// ---- GVLs/GVL10_VAR_PRG.TcGVL
(* Variables for program blocks *)
VAR_GLOBAL PERSISTENT
	
	nPowerFailureCounter					:UINT;
	
END_VAR
VAR_GLOBAL
	
	(* PLC start detected *)
	bFirstCycleDetected						:BOOL;
	bMachineSequenzAktiv					:BOOL;		(* PLC startup done (LED test) program in cyclic mode *)

	(* Clock generator *)
	bClock500ms								:BOOL;		(* Clock 500ms on/off *)
	bClock1s								:BOOL;		(* Clock 1s on/off *)
	bClock2s								:BOOL;		(* Clock 2s on/off *)
	bRisingEdge500ms						:BOOL;		(* Rising edge all 500ms over one cycle *)
	bRisingEdge1s							:BOOL;		(* Edge after 1s over a cycle *)
	bRisingEdge2s							:BOOL;		(* Edge after 2s over a cycle *)

END_VAR
(* End *)

// ---- GVLs/GVL20_Axis.TcGVL
(* GVL20_Axis - Global variables axis *)
{attribute 'TcContextName' := 'PlcTask'}
VAR_GLOBAL
	
(* Axis 1 inputs and outputs *)
	stAxis1									:AXIS_REF;

(* Axis 2 inputs and outputs *)
	stAxis2									:AXIS_REF;

(* Axis 3 - 4 (AX5203) inputs and outputs *)
	nAxis3TorqueFeedback			AT%I*	:INT;		(* Axis 3 current +/- 1000 *)
	nAxis4TorqueFeedback			AT%I*	:INT;		(* Axis 4 current +/- 1000 *)

	nAX5203DigitalInputs			AT%I*	:UINT;		(* Digital inputs AX5000
															BIT 0 - servo reference cam (axis 3)
															BIT 1 - servo reference cam (axis 4)
															BIT 2 - switch S26
															BIT 3 - switch S27 *)

	nAX5203DigitalOutputs			AT%Q*	:UINT;		(* Digital output AX5000 
															BIT 7 - Led H27 *)
	
	stAxis3									:AXIS_REF;
	stAxis4									:AXIS_REF;

(* Axis 5 (Handwheel) inputs and outputs *)
	stAxis5									:AXIS_REF;

END_VAR
(* End *)

// ---- GVLs/GVL30_DiagnosticEtherCAT.TcGVL
(* GVL30_DiagnosticEtherCAT *)
{attribute 'TcContextName' := 'PlcTask'}
VAR_GLOBAL

	fbDiagnosticEtherCAT					:FB_DiagnosticEtherCAT;

END_VAR
(* End *)

// ---- POUs/Sample OOP Conveyor/Device And Station Blocks/GVL_Products.TcGVL
VAR_GLOBAL
	arrParts : ARRAY[0..100] OF ST_PartData; // all the products currently in the machine
END_VAR

// ---- POUs/Sample UML SC/GVL_UML.TcGVL
VAR_GLOBAL
	nCounterInit				: INT;
	nCounterSaveInitSettings	: INT;
	nCounterClearXml			: INT;
	nCounterFillXml				: INT;
	nCounterSaveXml				: INT;
	nCounterClearText			: INT;
	nCounterFillText			: INT;
	nCounterSaveText			: INT;
	nCounterGetMasterID			: INT;
	nCounterGetClientID			: INT;
	nCounterSendToMaster		: INT;
	nCounterSendToClient		: INT;
	
	bMasterFirst				: BOOL;
	bClientFirst				: BOOL;
END_VAR

// ---- POUs/Sample OOP/Cylinder/ICylinder.TcIO
INTERFACE ICylinder

METHOD M_StateMachine : BOOL
VAR_INPUT
	bPosLeftReq  : BOOL;
	bPosRightReq : BOOL;
END_VAR
VAR_OUTPUT
	bAtLeftPos   : BOOL;
	bAtRightPos  : BOOL; 
END_VAR
END_METHOD

PROPERTY P_TimerValue : LREAL
GET
END_GET
SET
END_SET
END_PROPERTY

END_INTERFACE

// ---- POUs/Sample OOP/Regulator/IRegulator.TcIO
INTERFACE IRegulator

METHOD M_Active : UINT
VAR_INPUT
	(* controller input  *)
	fSetpointValue			: LREAL;		// setpoint value
	fActualValue			: LREAL;		// actual value
	bReset					: BOOL;			// reset flag
	(* controller values *)
	stRegParams				: ST_RegParams;
END_VAR
VAR_OUTPUT
	fCtrlOutput				: LREAL;		// controller output command
END_VAR
END_METHOD

PROPERTY P_Error : BOOL
GET
END_GET
SET
END_SET
END_PROPERTY

END_INTERFACE

// ---- POUs/Sample OOP/Table/Axis/IAxis.TcIO
INTERFACE IAxis

METHOD M_Diag : BOOL
VAR_INPUT
END_VAR
VAR_OUTPUT
	bNcError 	: BOOL;
	bDrvError 	: BOOL;
	iNcErrorId	: UDINT;
END_VAR
END_METHOD

METHOD M_Enable : BOOL
VAR_INPUT
	bEnable 	: BOOL;
	fOverride	: LREAL;
END_VAR
END_METHOD

METHOD M_HardwareDiag : BOOL
VAR_INPUT
	bExecute : BOOL;
END_VAR
END_METHOD

METHOD M_HardwareReset : BOOL
VAR_INPUT
	bExecute : BOOL;
END_VAR
END_METHOD

{attribute 'InstanceVar'}
METHOD M_Move : BOOL
VAR_INPUT
	bExecute	: BOOL;
	eMoveCmd	: E_MoveCmd;
	fVelocity	: LREAL;
	fPosition	: LREAL;
END_VAR
END_METHOD

METHOD M_Reset : BOOL
VAR_INPUT
	bExecute 	: BOOL;
END_VAR
END_METHOD

END_INTERFACE

// ---- POUs/Sample OOP Conveyor/Axis Blocks/I_Axis.TcIO
INTERFACE I_Axis

METHOD M_Disable : UDINT
VAR_INPUT
	bDisable : BOOL;
END_VAR
//The result of the method is an unsigned double integer
// 0 = idle 
// 1 = busy
// 3 = complete
// Any other number = Error
END_METHOD

METHOD M_Enable : UDINT
VAR_INPUT
	bEnable :BOOL;
END_VAR
//The result of the method is an unsigned double integer
// 0 = idle 
// 1 = busy
// 3 = complete
// Any other number = Error
END_METHOD

METHOD M_HardwareReset : UDINT
VAR_INPUT
	bReset:BOOL;
END_VAR
//The result of the method is an unsigned double integer
// 0 = idle 
// 1 = busy
// 3 = complete
// Any other number = Error number
END_METHOD

METHOD M_Jog : UDINT
VAR_INPUT
	bJogFwd : BOOL;
	bJogBwd : BOOL;
	fJogSpeed : LREAL;
END_VAR
//The result of the method is an unsigned double integer
// 0 = idle 
// 1 = busy
// 3 = complete
// Any other number = Error
END_METHOD

METHOD M_Reset : UDINT
VAR_INPUT
	bReset : BOOL;
END_VAR
//The result of the method is an unsigned double integer
// 0 = idle 
// 1 = busy
// 3 = complete
// Any other number = Error
END_METHOD

METHOD M_Speed : UDINT
VAR_INPUT
	bMoveVelocity : BOOL;
	fSpeed : LREAL;
END_VAR
//The result of the method is an unsigned double integer
// 0 = idle 
// 1 = busy
// 3 = complete
// Any other number = Error
END_METHOD

METHOD M_Stop : UDINT
VAR_INPUT
	bStop : BOOL;
END_VAR
//The result of the method is an unsigned double integer
// 0 = idle 
// 1 = busy
// 3 = complete
// Any other number = Error
END_METHOD

PROPERTY P_CurrentPosition : LREAL
GET
END_GET
SET
END_SET
END_PROPERTY

PROPERTY P_CurrentSpeed : LREAL
GET
END_GET
SET
END_SET
END_PROPERTY

PROPERTY P_Error : BOOL
GET
END_GET
SET
END_SET
END_PROPERTY

PROPERTY P_ErrorID : UDINT
GET
END_GET
SET
END_SET
END_PROPERTY

PROPERTY P_Ready : BOOL
GET
END_GET
SET
END_SET
END_PROPERTY

END_INTERFACE

// ---- POUs/Sample OOP Conveyor/Device And Station Blocks/I_Mode.TcIO
INTERFACE I_Mode

METHOD M_Auto : UDINT
VAR_INPUT
	bRequestAutoMode : BOOL;
END_VAR
END_METHOD

METHOD M_Disable : UDINT
VAR_INPUT
	bDisable : BOOL;
END_VAR
END_METHOD

METHOD M_Manual : UDINT
VAR_INPUT
	bRequestManualMode: BOOL;
END_VAR
END_METHOD

METHOD M_Reset : UDINT
VAR_INPUT
	bRequestReset:BOOL;
END_VAR
END_METHOD

PROPERTY P_CurrentState : E_Modes
GET
END_GET
SET
END_SET
END_PROPERTY

END_INTERFACE

// ---- POUs/RT Monitor/extMarksPrg.TcPOU
PROGRAM extMarksPrg
VAR
    fbLogMark	: FB_RTMon_LogMarkBase;	
	
	// user defined context
	idModule1 : UINT := 10001;	

		
	// Marks
	markCounter  : ST_RTMon_MarkDef := (nContextId := idModule1, nGroupId := 1, nEventId := 0); 
END_VAR

//fbLogMark.LogMarkEx(markCounter, TcMarkOption.Start OR TcMarkOption.RefToCaller);
IF GVL.fbCrititcalSection.Enter() THEN
	GVL.iGlobalCounter:=GVL.iGlobalCounter+1;
	ConsumeTime(50);
    GVL.fbCrititcalSection.Leave();
END_IF
//fbLogMark.LogMarkEx(markCounter, TcMarkOption.Stop OR TcMarkOption.RefToCaller);

END_PROGRAM

// ---- POUs/RT Monitor/logging/ConsumeTime.TcPOU
FUNCTION ConsumeTime : bool
VAR_INPUT
	DelayUs 	: UDINT;
END_VAR
VAR
	fbGetTime	: GETCPUACCOUNT;
	tStart		: UDINT;
	tNow		: UDINT;
END_VAR

fbGetTime(cpuAccountDW => tStart);
tNow := tStart;

WHILE (tNow - tStart) < DelayUs*10 DO
	fbGetTime(cpuAccountDW => tNow);
END_WHILE

END_FUNCTION

// ---- POUs/MainPOUs/MAIN.TcPOU
PROGRAM MAIN
(*******************************************************************************************************
Title				:	Main program 
Description			:	Calling the created subroutines (Task 1ms)
Version / Date		:	1.0.0 / 23.05.2016 / created program (Version progress see below)

Supported hardware	: 	Demo-Rack (LAGE version)

Used Documentation	:	
Documentation	
Version/Date 		:	

Required libraries 	: 	Please look in the "References" folder
********************************************************************************************************)
VAR
	
(* Cycle counter *)
	nCycleCounter							:UDINT;

(* act_SUps - 1s UPS - Uninterruptible power supply *)
	fbSUps									:FB_S_UPS_CX51x0 := (eUpsMode:=eSUPS_WrPersistData_Shutdown);
	bPowerFailDetect						:BOOL;

(* act_SystemStart *)
	eStateSystemStartSeq					:E_SystemStartupSequence;
	eSystemStartSeqErrStep					:E_SystemStartupSequence := eSystemStart_NoError;
	bSystemStartErr							:BOOL;
	bSystemStartEnd							:BOOL;
	fbTimerSystemStart						:TON;


(*******************************************************************************************************
Version / Date / Description:
1.0.0   / 23.05.2016 / created program
********************************************************************************************************)
(* End *)

	{attribute 'TcContextName':='PlcTask'}
	iCounter AT %Q*		: DINT;
	
	//fbMC2				: FB_MC2;
	//fbNCI				: FB_NCI;
	fbOOPAxisTable		: FB_OOPAxisTable;
	fbOOPCylReg			: FB_OOPCylinderRegulator;
	fbOOPConveyor		: FB_OOPConveyor;
	
	{attribute 'TcAnalytics'}
	fbScope				: FB_GenerateData;
	fbUmlSc				: FB_UML_SC_Composite;
	fbUmlSc_Lamp		: FB_UML_SC_Lamp;

	fbModeChangeTimer	: TON := (PT := T#60S);
	nRemainingModeTime	: UDINT;
	
	eSampleMode			: E_SampleMode;	
	eSampleModeMC2		: E_SampleMode;	
	eSampleModeNCI		: E_SampleMode;	
	eSampleModeOOP		: E_SampleMode;	
	eSampleModeOOPConv	: E_SampleMode;	

	nRadioButton		: INT;
	AxisRef				: ARRAY [1..iMAX_AXES_REF] OF AXIS_REF;			// axis reference (process data plc/nc)
	
	{attribute 'TcContextName':='PlcTask'}
	wFrmXWcState_MAIN AT %I*	: WORD; 			// link to NC-task related ethercat frame state (Frm0WcState)
	x1: WORD;
	
	fblog : FB_RTMon_LogMark;

END_VAR

(* MAIN - 1ms *)

(* THIS CODE IS ONLY AN EXAMPLE - YOU HAVE TO CHECK APTITUDE FOR YOUR APPLICATION *)

(* Cycle counter *)
	nCycleCounter := nCycleCounter + 1;


(* 1s USV *)
	act_SUps();


(* Startup detect *)
	IF TwinCAT_SystemInfoVarList._TaskInfo[GETCURTASKINDEXEX()].FirstCycle
	THEN
		bFirstCycleDetected	:= TRUE;
	END_IF


(* Startup- or machine sequence *)
	IF bFirstCycleDetected
	THEN
	(* Startup sequenz *)
		act_SystemStart();

		IF bSystemStartEnd
		THEN
			bFirstCycleDetected := FALSE;
			bMachineSequenzAktiv := TRUE;
		END_IF

	ELSIF bMachineSequenzAktiv
	THEN
	(* Machine sequenz *)
		(* Test general *)
			GeneralPlc();
		
		(* Test blinker *)
			Blinker();

		(* Test clock generator *)
			ClockGenerator();
		
		(* Test axis *)
			AxisGeneral();
			Axis1();
			Axis2();
			Axis3();
			Axis4();
			stAxis5.ReadStatus();

		(* Test EtherCAT diacnostic *)
			DiagnosticEtherCAT();
			
		(* Test - XFC - extrem fast control *)	
			DcTimes();
			AnalogOutputOversampling();
			PositionCamTimeStampAxis2();
			SignalLengthMeasurementCamAxis2();
			TouchProbeTimeStampCamAxis2();

		(* Test TwinSAFE *)	
			TwinSAFE();
		
	END_IF

(* End *)

iCounter := iCounter + 1;

//switch mode (MC2, NCI, OOP)
A_ModeSwitch();

(*//call MC2 sample
fblog.LogStart(1,0); //added this
fbMC2(AxisRef := AxisRef, eSampleModeIn := eSampleMode, eSampleModeOut => eSampleModeMC2);
fblog.LogStop(1,0); // added this*)


//call NCI sample
fblog.LogStart(2,0); //added this
NCI();
//fbNCI(AxisRef := AxisRef, eSampleModeIn := eSampleMode, eSampleModeOut => eSampleModeNCI);
fblog.LogStop(2,0);

//Call Cam Table Sample
CamTable();

//Call External Setpoint Generator Sample
Ext_SP_Gen();

//call OOP sample
fblog.LogStart(3,0);
fbOOPAxisTable(AxisRef := AxisRef, eSampleModeIn := eSampleMode, eSampleModeOut => eSampleModeOOP);
fbOOPCylReg();
fblog.LogStop(3,0);

//call OOP conveyor sample
fblog.logstart(4,0);
fbOOPConveyor(AxisRef := AxisRef, eSampleModeIn := eSampleMode, eSampleModeOut => eSampleModeOOPConv);
fblog.logstop(4,0);

//call language samples
fblog.LogMark(5,0);
MAIN_CFC();					//continuous flow chart
fblog.LogMark(5,1);
MAIN_CFC_PageOriented();	//continuous flow chart, page oriented
fblog.LogMark(5,2);
MAIN_FBD_IL_LD();			//use language switching via menu "FBD/IL/LD, function block diagram, instruction list, ladder logic 
fblog.LogMark(5,3);
MAIN_SFC();					//sequential flow chart 
fblog.LogMark(5,4);
MAIN_ST();					//structured text
fblog.LogStop(5,0);


//call UML SC composite sample
fblog.LogStart(6,0);
fbUmlSc();
fbUmlSc_Lamp();
fblog.LogStop(6,0);

x1 := wFrmXWcState_MAIN;

//Call TwinSAFE Program
TwinSAFE();

//Call IoT Program
IoT_JSON_XML();

//Call Database Server Sample
CSVSample();

ACTION A_ModeSwitch:
//decide for an active motion sample
fbModeChangeTimer(IN := TRUE);
nRemainingModeTime := TIME_TO_UDINT(fbModeChangeTimer.PT-fbModeChangeTimer.ET)/1000;

IF fbModeChangeTimer.Q OR (eSampleMode = eSMode_Idle) OR (nRadioButton > 0) THEN
	//switch if ready 
	
	IF (eSampleModeMC2 = eSMode_Idle) AND (eSampleModeNCI = eSMode_Idle) AND (eSampleModeOOP = eSMode_Idle) AND (eSampleModeOOPConv = eSMode_Idle) THEN
		//ready to switch
		fbModeChangeTimer(IN := FALSE);
		
		CASE eSampleMode OF
		eSMode_Idle:
			CASE nRadioButton OF
			1:
				eSampleMode := eSMode_MC2_Req;
			2:			
				eSampleMode := eSMode_NCI_Req;
			3:			
				eSampleMode := eSMode_OOP_Req;
			4:			
				eSampleMode := eSMode_OOPConv_Req;
			ELSE //idle
				eSampleMode := eSMode_MC2_Req;
			END_CASE
			
		eSMode_MC2_Req:
			CASE nRadioButton OF
			1:
				eSampleMode := eSMode_MC2_Req;
			2:			
				eSampleMode := eSMode_NCI_Req;
			3:			
				eSampleMode := eSMode_OOP_Req;
			4:			
				eSampleMode := eSMode_OOPConv_Req;
			ELSE //idle
				eSampleMode := eSMode_NCI_Req;
			END_CASE
			
		eSMode_NCI_Req:
			CASE nRadioButton OF
			1:
				eSampleMode := eSMode_MC2_Req;
			2:			
				eSampleMode := eSMode_NCI_Req;
			3:			
				eSampleMode := eSMode_OOP_Req;
			4:			
				eSampleMode := eSMode_OOPConv_Req;
			ELSE //idle
				eSampleMode := eSMode_OOP_Req;
			END_CASE
			
		eSMode_OOP_Req:
			CASE nRadioButton OF
			1:
				eSampleMode := eSMode_MC2_Req;
			2:			
				eSampleMode := eSMode_NCI_Req;
			3:			
				eSampleMode := eSMode_OOP_Req;
			4:			
				eSampleMode := eSMode_OOPConv_Req;
			ELSE //idle
				eSampleMode := eSMode_MC2_Req;
			END_CASE
			
		eSMode_OOPConv_Req:
			CASE nRadioButton OF
			1:
				eSampleMode := eSMode_MC2_Req;
			2:			
				eSampleMode := eSMode_NCI_Req;
			3:			
				eSampleMode := eSMode_OOP_Req;
			4:			
				eSampleMode := eSMode_OOPConv_Req;
			ELSE //idle
				eSampleMode := eSMode_MC2_Req;
			END_CASE
			
		ELSE
			eSampleMode := eSMode_MC2_Req;
		END_CASE
		
		nRadioButton := 0;
	END_IF 
END_IF
END_ACTION

ACTION act_SUps:
(* Aktion - 1s UPS - Uninterruptible power supply *)

	fbSUps(); (* see instance declaration for initalisation of eUpsMode parameter *) 

	(*
	Default Values of FB_S_UPS_CX51x0-Inputs:
						sNetID 			:=	'' -> local netid
						iPLCPort 		:=	AMSPORT_R0_PLC_RTS1 -> 801 = 1st PLC Runtime 
						iUPSPort		:=	16#588 -> Port for reading Power State of UPS
						tTimeout 		:=	DEFAULT_ADS_TIMEOUT -> 5S
						eUpsMode 		:=	eSUPS_WrPersistData_Shutdown -> writing persistent data + shutdown
						ePersistentMode :=	SPDM_2PASS -> All data is from same plc cycle, cycletime exceeds possible. Plc stops with the shutdown, a few cycles after writing persistent data. 
						tRecoverTime 	:=	T#10s -> 10s power to recover from short power failure before eSUPS_PowerOK is reported (in mode eSUPS_WrPersistData_NoShutdown/eSUPS_CheckPowerStatus)

	eUpsMode =							in case of powerfailure:
	 	eSUPS_WrPersistData_Shutdown 	->	writing of persistent data + shutdown
	 	eSUPS_WrPersistData_NoShutdown 	->	writing of PERSISTENT data, no shutdown
	 	eSUPS_CheckPowerStatus 			->	reports powerfailure without ACTION (no writing, no shutdown) 
	 	eSUPS_ImmediateShutdown 		->	skips writing of data, immediate shutdown
	*)	

(* Power fail detected *)
	IF fbSUps.bPowerFailDetect
		AND NOT bPowerFailDetect
	THEN
	
		(* Count the power failures *)
		nPowerFailureCounter := nPowerFailureCounter + 1;
		bPowerFailDetect	 := TRUE;
	
	ELSE

		IF NOT fbSUps.bPowerFailDetect
		THEN
			bPowerFailDetect:=FALSE;
		END_IF

	END_IF

(* End *)
END_ACTION

ACTION act_SystemStart:
(* Aktion system start *)

	CASE eStateSystemStartSeq OF

	
		eSystemStart_Start			: 	(* Waiting for start *)
		
				eStateSystemStartSeq := eSystemStart_Init;

				
		eSystemStart_Init			:	(* Initialize *)

				fbTimerSystemStart(IN := FALSE);
				eStateSystemStartSeq := eSystemStart_LedOn;

				
		eSystemStart_LedOn			:	(* Sequence Leds on *)

				fbTimerSystemStart(	
					IN := TRUE,
					PT := T#2250MS);

				bLedH10	:=	fbTimerSystemStart.ET > T#250MS;
				bLedH20 :=  bLedH10;
				bLedH31 :=  bLedH10;
				bLedH11	:=	fbTimerSystemStart.ET > T#500MS;
				bLedH21 :=  bLedH11;
				bLedH32 :=  bLedH11;
				bLedH12	:=	fbTimerSystemStart.ET > T#750MS;
				bLedH22 :=  bLedH12;
				bLedH33 :=  bLedH12;
				bLedH13	:=	fbTimerSystemStart.ET > T#1000MS;
				bLedH23 :=  bLedH13;
				bLedH14	:=	fbTimerSystemStart.ET > T#1250MS;
				bLedH24 :=  bLedH14;
				bLedH15	:=	fbTimerSystemStart.ET > T#1500MS;
				bLedH25 :=  bLedH15;
				bLedH16	:=	fbTimerSystemStart.ET > T#1750MS;
				bLedH26 :=  bLedH16;
				bLedH17	:=	fbTimerSystemStart.ET > T#2000MS;
				nAX5203DigitalOutputs.7 :=  bLedH17;

				IF fbTimerSystemStart.Q
				THEN
					fbTimerSystemStart(IN := FALSE);
					eStateSystemStartSeq := eSystemStart_LedOff;
				ELSIF FALSE
				THEN
					(* If error then notice the step *)
					eSystemStartSeqErrStep := eStateSystemStartSeq;
					eStateSystemStartSeq   := eSystemStart_ErrorStep;
				END_IF

				
		eSystemStart_LedOff			:	(* Sequence Leds off *)

				fbTimerSystemStart(	
					IN := TRUE,
					PT := T#2250MS);

				bLedH10	:=	fbTimerSystemStart.ET < T#250MS;
				bLedH20 :=  bLedH10;
				bLedH31 :=  bLedH10;
				bLedH11	:=	fbTimerSystemStart.ET < T#500MS;
				bLedH21 :=  bLedH11;
				bLedH32 :=  bLedH11;
				bLedH12	:=	fbTimerSystemStart.ET < T#750MS;
				bLedH22 :=  bLedH12;
				bLedH33 :=  bLedH12;
				bLedH13	:=	fbTimerSystemStart.ET < T#1000MS;
				bLedH23 :=  bLedH13;
				bLedH14	:=	fbTimerSystemStart.ET < T#1250MS;
				bLedH24 :=  bLedH14;
				bLedH15	:=	fbTimerSystemStart.ET < T#1500MS;
				bLedH25 :=  bLedH15;
				bLedH16	:=	fbTimerSystemStart.ET < T#1750MS;
				bLedH26 :=  bLedH16;
				bLedH17	:=	fbTimerSystemStart.ET < T#2000MS;
				nAX5203DigitalOutputs.7 :=  bLedH17;
									
				IF fbTimerSystemStart.Q
				THEN
					eStateSystemStartSeq := eSystemStart_Done;
				ELSIF FALSE
				THEN
					(* If error then notice the step *)
					eSystemStartSeqErrStep := eStateSystemStartSeq;
					eStateSystemStartSeq   := eSystemStart_ErrorStep;
				END_IF

				
		eSystemStart_Done			:	(* System start done *)

				bSystemStartEnd := TRUE;

				
		eSystemStart_ErrorStep		:	(* Error on system start *)

				bSystemStartErr := TRUE;

				IF FALSE
				THEN
					bSystemStartErr        := FALSE;
					eSystemStartSeqErrStep := eSystemStart_NoError;
					eStateSystemStartSeq   := eSystemStart_Start;
				END_IF 

	ELSE
		
		(* If not a valid step is active, then put on start *)
		eSystemStartSeqErrStep := eSystemStart_NoError;
		eStateSystemStartSeq   := eSystemStart_Start;
	
	END_CASE

(* End *)
END_ACTION

END_PROGRAM

// ---- POUs/Sample OOP/FB_OOPAxisTable.TcPOU
FUNCTION_BLOCK FB_OOPAxisTable
VAR_INPUT
	eSampleModeIn	: E_SampleMode;	
END_VAR
VAR_IN_OUT
	AxisRef			: ARRAY [1..iMAX_AXES_REF] OF AXIS_REF;			// axis reference (process data plc/nc)
END_VAR
VAR_OUTPUT
	eSampleModeOut	: E_SampleMode;	
END_VAR
VAR
	iCounter 			: DINT;
END_VAR	
VAR
	//instances of axes FBs (of type FB_NcAxes or derived from FB_NcAxis, like AX5000, Servo Termins, Stepper, DC, ...)
	fbAX5000Axis1	: FB_AX5000Axis;
	fbAX5000Axis2	: FB_AX5000Axis;
	fbNcAxis		: FB_NcAxis;
		
	//interface pointers
	ipAxisX			: IAxis;
	ipAxisY			: IAxis;
	ipAxisZ			: IAxis;

	//device
	fbTable			: FB_Table;
	bExecute		: BOOL;
	bBusy			: BOOL;
	
	Timer			: TON := (PT := T#3s);
END_VAR

iCounter := iCounter + 1;

IF (eSampleModeIn = eSMode_OOP_Req) OR (eSampleModeOut = eSMode_OOP_Act) THEN
	//assign axes instances to the interface pointers
	ipAxisX := fbAX5000Axis1;
	ipAxisY := fbAX5000Axis2;
	ipAxisZ	:= fbNcAxis;
	
	//call axes with their axes references
	fbAX5000Axis1(sAxis	:= AxisRef[1]);
	fbAX5000Axis2(sAxis	:= AxisRef[2]);
	fbNcAxis(sAxis	:= AxisRef[3]);
	
	Timer(IN := TRUE);
	IF Timer.Q THEN
		Timer(IN := FALSE);
		bExecute := TRUE;
	END_IF
	
	//call device that uses axes via interface, therefore the axis type does not matter anymore
	fbTable(
		fbServoAxisX := ipAxisX,
		fbServoAxisY := ipAxisY,
		fbServoAxisZ := ipAxisZ,
		bExecute	 := bExecute,
		bBusy		 => bBusy
	);
		
	bExecute := FALSE;

	IF bBusy THEN
		eSampleModeOut := eSMode_OOP_Act;
	ELSE
		eSampleModeOut := eSMode_Idle;
	END_IF
END_IF

END_FUNCTION_BLOCK

// ---- POUs/Sample OOP/Table/Axis/FB_AX5000Axis.TcPOU
FUNCTION_BLOCK FB_AX5000Axis EXTENDS FB_NcAxis
VAR_INPUT
END_VAR
VAR_OUTPUT
END_VAR
VAR
	fbSoEReadDiagNumber : FB_SoEReadDiagNumber;
	iDiagNumber			: UDINT;
	fbSoEReset			: FB_SoEReset;
END_VAR

METHOD M_HardwareDiag : BOOL
VAR_INPUT
	bExecute	: BOOL;
END_VAR
//get hardware diag
CASE eCurState OF
eAxisState_Idle:
	IF bExecute AND NOT bExecHWDiag_  THEN
		fbSoEReadDiagNumber(
			NetId:= '', 
			Execute:= TRUE, 
			Axis:= sAxis, 
		);
		eCurState := eAxisState_Diag;
	END_IF

eAxisState_Diag:
	fbSoEReadDiagNumber(
		NetId:= '', 
		Execute:= TRUE, 
		Axis:= sAxis, 
	);
	IF NOT fbSoEReadDiagNumber.Busy  THEN
		fbSoEReadDiagNumber(
			Execute:= FALSE, 
			Axis:= sAxis, 
			DiagNumber=> iDiagNumber
		);
		eCurState := eAxisState_Idle;
	END_IF
	
END_CASE

M_HardwareDiag 	:= eCurState <> eAxisState_Idle;	
bExecHWDiag_	:= bExecute;
END_METHOD

METHOD M_HardwareReset : BOOL
VAR_INPUT
	bExecute	: BOOL;
END_VAR
//reset axis
CASE eCurState OF
eAxisState_Idle:
	IF bExecute AND NOT bExecHWRes_ THEN
		fbSoEReset(
			NetId:= '', 
			Execute:= TRUE, 
			Axis:= sAxis, 
		);
		eCurState := eAxisState_Reset;
	END_IF

eAxisState_Reset:
	fbSoEReset(
		NetId:= '', 
		Execute:= TRUE, 
		Axis:= sAxis, 
	);
	IF NOT fbSoEReset.Busy THEN
		fbSoEReset(
			Execute:= FALSE, 
			Axis:= sAxis, 
		);
		eCurState := eAxisState_Idle;
	END_IF

END_CASE

M_HardwareReset := eCurState <> eAxisState_Idle;	
bExecHWRes_		:= bExecute;
END_METHOD

END_FUNCTION_BLOCK

// ---- POUs/Sample OOP/Table/Axis/FB_NcAxis.TcPOU
FUNCTION_BLOCK FB_NcAxis IMPLEMENTS IAxis
VAR_IN_OUT
	sAxis		: AXIS_REF;
END_VAR
VAR_INPUT
END_VAR
VAR_OUTPUT
	bActive		: BOOL;
	bBusy		: BOOL;
	bDone		: BOOL;
	bError		: BOOL;
	iErrorId	: UDINT;
	eCurState	: E_AxisState;
END_VAR
VAR
	//PLCopen FBs for axes
	fbMcPower	: MC_Power;
	fbMcReset	: MC_Reset;
	fbMcMoveAbs	: MC_MoveAbsolute;
	fbMcMoveMod	: MC_MoveModulo;
	fbMcMoveRel	: MC_MoveRelative;
	fbMcMoveVel	: MC_MoveVelocity;

	//rising edge detection
	bExecMove_	: BOOL;
	bExecHWDiag_: BOOL;
	bExecHWRes_	: BOOL;
	bExecReset_	: BOOL;
END_VAR

;

METHOD M_Diag : BOOL
VAR_INPUT
END_VAR
VAR_OUTPUT
	bNcError 	: BOOL;
	bDrvError 	: BOOL;
	iNcErrorId	: UDINT;
END_VAR
//get axis diag
sAxis.ReadStatus();
bNcError	:= sAxis.NcToPlc.StateDWord.31;
bDrvError	:= sAxis.NcToPlc.StateDWord.28;
iNcErrorId	:= sAxis.NcToPlc.ErrorCode;
M_Diag 		:= bNcError OR bDrvError OR (iNcErrorId <> 0);
END_METHOD

METHOD M_Enable : BOOL
VAR_INPUT
	bEnable		: BOOL;
	fOverride	: LREAL;
END_VAR
//enable axis
fbMcPower(
	Enable		:= bEnable, 	Enable_Positive	:= bEnable,	Enable_Negative	:= bEnable, 
	Override	:= fOverride, 	Axis			:= sAxis
);
M_Enable := fbMcPower.Status;
END_METHOD

METHOD M_HardwareDiag : BOOL
VAR_INPUT
	bExecute	: BOOL;
END_VAR
//get hardware diag --> overwrite method if necessary
CASE eCurState OF
eAxisState_Idle:
	IF bExecute AND NOT bExecHWDiag_ THEN
		eCurState := eAxisState_Diag;
	END_IF

eAxisState_Diag:
		eCurState := eAxisState_Idle;

END_CASE

M_HardwareDiag 	:= eCurState <> eAxisState_Idle;	
bExecHWDiag_	:= bExecute;
END_METHOD

METHOD M_HardwareReset : BOOL
VAR_INPUT
	bExecute	: BOOL;
END_VAR
//hardware reset axis --> overwrite method if necessary
CASE eCurState OF
eAxisState_Idle:
	IF bExecute AND NOT bExecHWRes_ THEN
		eCurState := eAxisState_Reset;
	END_IF

eAxisState_Reset:
		eCurState := eAxisState_Idle;

END_CASE

M_HardwareReset := eCurState <> eAxisState_Idle;	
bExecHWRes_		:= bExecute;
END_METHOD

METHOD M_Move : BOOL
VAR_INPUT
	bExecute	: BOOL;
	eMoveCmd	: E_MoveCmd;
	fVelocity	: LREAL;
	fPosition	: LREAL;
END_VAR
//move axis
CASE eCurState OF
eAxisState_Idle:	
	IF bExecute AND NOT bExecMove_ THEN
		CASE eMoveCmd OF
		eCmd_MoveAbsolute:
			fbMcMoveAbs(
				Execute	:= bExecute, 	Position:= fPosition,	Velocity:= fVelocity, 
				Axis	:= sAxis, 		Done	=> bDone,		Busy	=> bBusy, 
				Active	=> bActive, 	Error	=> bError,		ErrorID	=> iErrorId
			);
			eCurState := eAxisState_Move;
		
		eCmd_MoveModulo:
			fbMcMoveMod(
				Execute	:= bExecute, 	Position:= fPosition,	Velocity:= fVelocity, 
				Axis	:= sAxis, 		Done	=> bDone, 		Busy	=> bBusy, 
				Active	=> bActive, 	Error	=> bError,		ErrorID	=> iErrorId
			);
			eCurState := eAxisState_Move;
		
		eCmd_MoveRelative:
			fbMcMoveRel(
				Execute	:= bExecute, 	Distance:= fPosition,	Velocity:= fVelocity, 
				Axis	:= sAxis, 		Done	=> bDone,		Busy	=> bBusy, 
				Active	=> bActive, 	Error	=> bError,		ErrorID	=> iErrorId
			);
			eCurState := eAxisState_Move;
		
		eCmd_MoveVelocity:
			fbMcMoveVel(
				Execute	:= bExecute, 	Velocity:= fVelocity,	Axis	:= sAxis, 
				InVelocity=> bDone,		Busy	=> bBusy,		Active	=> bActive, 
				Error	=> bError, 		ErrorID	=> iErrorId,	Busy	=> bBusy,
				Active	=> bActive,		Error	=> bError,		ErrorID	=> iErrorId
			);		
			eCurState := eAxisState_Move;
		END_CASE
	END_IF
		
eAxisState_Move:
	CASE eMoveCmd OF
	eCmd_MoveAbsolute:
		fbMcMoveAbs(
			Execute	:= TRUE, 		Position:= fPosition,	Velocity:= fVelocity, 
			Axis	:= sAxis, 		Done	=> bDone,		Busy	=> bBusy, 
			Active	=> bActive, 	Error	=> bError, 		ErrorID	=> iErrorId
		);
		IF bDone OR bError THEN
			fbMcMoveAbs(Execute	:= FALSE,Axis := sAxis); 
			eCurState := eAxisState_Idle;
		END_IF
	
	eCmd_MoveModulo:
		fbMcMoveMod(
			Execute	:= TRUE, 		Position:= fPosition,	Velocity:= fVelocity, 
			Axis	:= sAxis, 		Done	=> bDone,		Busy	=> bBusy, 
			Active	=> bActive, 	Error	=> bError,		ErrorID	=> iErrorId
		);
		IF bDone OR bError THEN
			fbMcMoveMod(Execute	:= FALSE,Axis := sAxis); 
			eCurState := eAxisState_Idle;
		END_IF
	
	eCmd_MoveRelative:
		fbMcMoveRel(
			Execute	:= TRUE, 		Distance:= fPosition,	Velocity:= fVelocity, 
			Axis	:= sAxis, 		Done	=> bDone,		Busy	=> bBusy, 
			Active	=> bActive, 	Error	=> bError,		ErrorID	=> iErrorId
		);
		IF bDone OR bError THEN
			fbMcMoveRel(Execute	:= FALSE,Axis := sAxis); 
			eCurState := eAxisState_Idle;
		END_IF
	
	eCmd_MoveVelocity:
		fbMcMoveVel(
			Execute	:= TRUE, 		Velocity:= fVelocity,	Axis	:= sAxis, 
			InVelocity=> bDone,		Busy	=> bBusy,		Active	=> bActive, 
			Error	=> bError, 		ErrorID	=> iErrorId,	Busy	=> bBusy, 		
			Active	=> bActive,		Error	=> bError,		ErrorID	=> iErrorId
		);		
		IF bDone OR bError THEN
			fbMcMoveVel(Execute	:= FALSE,Axis := sAxis); 
			eCurState := eAxisState_Idle;
		END_IF
	END_CASE
END_CASE

M_Move 		:= (eCurState <> eAxisState_Idle);
bExecMove_	:= bExecute;
END_METHOD

METHOD M_Reset : BOOL
VAR_INPUT
	bExecute	: BOOL;
END_VAR
//reset nc axis
CASE eCurState OF
eAxisState_Idle:
	IF bExecute AND NOT bExecReset_ THEN
		fbMcReset(
			Execute	:= bExecute, 	Axis	:= sAxis,	Done	=> bDone, 
			Busy	=> bBusy, 		Error	=> bError,	ErrorID	=> iErrorId 
		);
		eCurState := eAxisState_Reset;
	END_IF

eAxisState_Reset:
	fbMcReset(
		Execute	:= FALSE, 	Axis	:= sAxis,	Done	=> bDone, 
		Busy	=> bBusy, 	Error	=> bError,	ErrorID	=> iErrorId 
	);
	IF fbMcReset.Done OR fbMcReset.Error THEN
		eCurState := eAxisState_Idle;
	END_IF
END_CASE

M_Reset 	:= eCurState <> eAxisState_Idle;	
bExecReset_	:= bExecute;
END_METHOD

END_FUNCTION_BLOCK

// ---- POUs/Sample OOP/Table/FB_Table.TcPOU
FUNCTION_BLOCK FB_Table
VAR_IN_OUT
	fbServoAxisX	: IAxis; //Pass the reference to ANY block that uses FB_NcAxis as a base class
	fbServoAxisY	: IAxis; //Pass the reference to ANY block that uses FB_NcAxis as a base class
	fbServoAxisZ	: IAxis; //Pass the reference to ANY block that uses FB_NcAxis as a base class
END_VAR
VAR_INPUT
	bEnable			: BOOL	:= TRUE;
	fOverride		: LREAL	:= 100;
	bExecute		: BOOL;
END_VAR
VAR_OUTPUT
	bEnabled		: BOOL;
	bBusy			: BOOL;
	bError			: BOOL;
END_VAR
VAR
	iState			: INT;
	bExecute_		: BOOL;

	eCurStateAxisX	: E_AxisState;
	bEnabledAxisX	: BOOL;
	bBusyAxisX		: BOOL;
	bErrorAxisX		: BOOL;

	eCurStateAxisY	: E_AxisState;
	bEnabledAxisY	: BOOL;
	bBusyAxisY		: BOOL;
	bErrorAxisY		: BOOL;

	eCurStateAxisZ	: E_AxisState;
	bEnabledAxisZ	: BOOL;
	bBusyAxisZ		: BOOL;
	bErrorAxisZ		: BOOL;
END_VAR

//NC axes can be used independent of axes type (AX5000, stepper, analog axis, ...) incl. hardware reset and diagnostic  

//enable axes
bEnabledAxisX 	:= fbServoAxisX.M_Enable(bEnable:= bEnable, fOverride:= fOverride);
bEnabledAxisY 	:= fbServoAxisY.M_Enable(bEnable:= bEnable, fOverride:= fOverride);
bEnabledAxisZ 	:= fbServoAxisZ.M_Enable(bEnable:= bEnable, fOverride:= fOverride);
bEnabled		:= bEnabledAxisX AND bEnabledAxisY AND bEnabledAxisZ;

//check for cyclic diagnostics
bErrorAxisX		:= fbServoAxisX.M_Diag();
bErrorAxisY		:= fbServoAxisY.M_Diag();
bErrorAxisZ		:= fbServoAxisZ.M_Diag();
bError			:= bError OR bErrorAxisX OR bErrorAxisY OR bErrorAxisZ;

//state machine
CASE iState OF
	0:	//idle state
		IF (bExecute AND NOT bExecute_) THEN
			IF bError THEN
				iState := 10;
			ELSIF bEnabled THEN
				iState := iState + 1;
			END_IF
		END_IF	
		
	1:	//move x 200, y 200, z 200
		bBusyAxisX := fbServoAxisX.M_Move(bExecute:= TRUE, eMoveCmd:= eCmd_MoveAbsolute, fVelocity:= 100.0, fPosition:= 200.0);
		bBusyAxisY := fbServoAxisY.M_Move(bExecute:= TRUE, eMoveCmd:= eCmd_MoveAbsolute, fVelocity:= 100.0, fPosition:= 200.0);
		bBusyAxisZ := fbServoAxisZ.M_Move(bExecute:= TRUE, eMoveCmd:= eCmd_MoveAbsolute, fVelocity:= 100.0, fPosition:= 200.0);
		IF NOT bBusyAxisX AND NOT bBusyAxisY AND NOT bBusyAxisZ THEN
			bBusyAxisX := fbServoAxisX.M_Move(bExecute:= FALSE, eMoveCmd:= eCmd_MoveAbsolute, fVelocity:= 100.0, fPosition:= 200.0);
			bBusyAxisY := fbServoAxisY.M_Move(bExecute:= FALSE, eMoveCmd:= eCmd_MoveAbsolute, fVelocity:= 100.0, fPosition:= 200.0);
			bBusyAxisZ := fbServoAxisZ.M_Move(bExecute:= FALSE, eMoveCmd:= eCmd_MoveAbsolute, fVelocity:= 100.0, fPosition:= 200.0);
			iState := iState + 1;
		END_IF
		
	2:	//move x 100, y 300
		bBusyAxisX := fbServoAxisX.M_Move(bExecute:= TRUE, eMoveCmd:= eCmd_MoveAbsolute, fVelocity:= 150.0, fPosition:= 100.0);
		bBusyAxisY := fbServoAxisY.M_Move(bExecute:= TRUE, eMoveCmd:= eCmd_MoveAbsolute, fVelocity:= 150.0, fPosition:= 300.0);
		IF NOT bBusyAxisX AND NOT bBusyAxisY THEN
			bBusyAxisX := fbServoAxisX.M_Move(bExecute:= FALSE, eMoveCmd:= eCmd_MoveAbsolute, fVelocity:= 150.0, fPosition:= 100.0);
			bBusyAxisY := fbServoAxisY.M_Move(bExecute:= FALSE, eMoveCmd:= eCmd_MoveAbsolute, fVelocity:= 150.0, fPosition:= 300.0);
			iState := iState + 1;
		END_IF
		
	3:	//move x 0, y 0, z 0
		bBusyAxisX := fbServoAxisX.M_Move(bExecute:= TRUE, eMoveCmd:= eCmd_MoveAbsolute, fVelocity:= 50.0, fPosition:= 0.0);
		bBusyAxisY := fbServoAxisY.M_Move(bExecute:= TRUE, eMoveCmd:= eCmd_MoveAbsolute, fVelocity:= 150.0, fPosition:= 0.0);
		bBusyAxisZ := fbServoAxisZ.M_Move(bExecute:= TRUE, eMoveCmd:= eCmd_MoveAbsolute, fVelocity:= 150.0, fPosition:= 0.0);
		IF NOT bBusyAxisX AND NOT bBusyAxisY AND NOT bBusyAxisZ THEN
			bBusyAxisX := fbServoAxisX.M_Move(bExecute:= FALSE, eMoveCmd:= eCmd_MoveAbsolute, fVelocity:= 50.0, fPosition:= 0.0);
			bBusyAxisY := fbServoAxisY.M_Move(bExecute:= FALSE, eMoveCmd:= eCmd_MoveAbsolute, fVelocity:= 150.0, fPosition:= 0.0);
			bBusyAxisZ := fbServoAxisZ.M_Move(bExecute:= FALSE, eMoveCmd:= eCmd_MoveAbsolute, fVelocity:= 150.0, fPosition:= 0.0);
			iState := 0;
		END_IF
		
	10:	//hardware diag
		bBusyAxisX := fbServoAxisX.M_HardwareDiag(bExecute:= TRUE);
		bBusyAxisY := fbServoAxisY.M_HardwareDiag(bExecute:= TRUE);
		bBusyAxisZ := fbServoAxisZ.M_HardwareDiag(bExecute:= TRUE);
		IF NOT bBusyAxisX AND NOT bBusyAxisY AND NOT bBusyAxisZ THEN
			bBusyAxisX := fbServoAxisX.M_HardwareDiag(bExecute:= FALSE);
			bBusyAxisY := fbServoAxisY.M_HardwareDiag(bExecute:= FALSE);
			bBusyAxisZ := fbServoAxisZ.M_HardwareDiag(bExecute:= FALSE);
			iState := iState + 1;
		END_IF

	11:	//hardware reset
		bBusyAxisX := fbServoAxisX.M_HardwareReset(bExecute:= TRUE);
		bBusyAxisY := fbServoAxisY.M_HardwareReset(bExecute:= TRUE);
		bBusyAxisZ := fbServoAxisZ.M_HardwareReset(bExecute:= TRUE);
		IF NOT bBusyAxisX AND NOT bBusyAxisY AND NOT bBusyAxisZ THEN
			bBusyAxisX := fbServoAxisX.M_HardwareReset(bExecute:= FALSE);
			bBusyAxisY := fbServoAxisY.M_HardwareReset(bExecute:= FALSE);
			bBusyAxisZ := fbServoAxisZ.M_HardwareReset(bExecute:= FALSE);
			iState := iState + 1;
		END_IF
		
	12:	//nc reset
		bBusyAxisX := fbServoAxisX.M_Reset(bExecute:= TRUE);
		bBusyAxisY := fbServoAxisY.M_Reset(bExecute:= TRUE);
		bBusyAxisZ := fbServoAxisZ.M_Reset(bExecute:= TRUE);
		IF NOT bBusyAxisX AND NOT bBusyAxisY AND NOT bBusyAxisZ THEN
			bBusyAxisX := fbServoAxisX.M_Reset(bExecute:= FALSE);
			bBusyAxisY := fbServoAxisY.M_Reset(bExecute:= FALSE);
			bBusyAxisZ := fbServoAxisZ.M_Reset(bExecute:= FALSE);
			bError := FALSE;
			iState := 0;
		END_IF

END_CASE

bBusy		:= bBusyAxisX OR bBusyAxisY OR bBusyAxisZ;
bExecute_ 	:= bExecute;

END_FUNCTION_BLOCK

// ---- POUs/Sample OOP/FB_OOPCylinderRegulator.TcPOU
FUNCTION_BLOCK FB_OOPCylinderRegulator
VAR
	iCounter 				: DINT;	

	(* Interface Instance of ICylinder *)
	ipCylinder 				: ICylinder;

	(* cylinder with feedback and without/with diag  *)
	fbCylinder 				: FB_Cylinder;		//instance of cylinder without diag 
	fbCylinderDiag			: FB_CylinderDiag;	//instance of cylinder with diag
	bEnableDiag				: BOOL := FALSE;	//enable diagnose cylinder
	bDiagAvailable			: BOOL;				//diag is enabled
	lrTimerValue 			: LREAL := 0.2;		//simulation time [s]
	tTimeOutDiag 			: TIME := T#1S100MS;//diagnose timeout
	bDiag	 				: BOOL;				//diagnose feedback

	(* cmds/state *)
	bMoveToLeftReq AT %I*	: BOOL;		//cmd move to left side
	bMoveToRightReq AT %I*	: BOOL;		//cmd move to right side
	bCylinderAtLeft AT %Q* 	: BOOL;		//state at left side
	bCylinderAtRight AT %Q*	: BOOL;		//state at left side


	(* Interface Instance of IRegulator *)
	ipRegulator 		: IRegulator;

	(* P/PID Regulator *)
	fbBasicP			: FB_BasicP;		// instance of P-Controller
	fbBasicPID			: FB_BasicPID;		// instance of PID-Controller
	bEnablePID			: BOOL;				// enable PID
	bPIDEnabled			: BOOL;				// PID enabled
	fSetpointValue		: LREAL;			// setpoint value
	fActualValue		: LREAL;			// actual value
	bReset				: BOOL;				// reset flag
	stRegParams			: ST_RegParams;		// parameters for the regulator
	fCtrlOutput			: LREAL;			// controller output command
	bErrorFlag			: BOOL;				// controller error
	

	(* common *)
	Timer 				: TON := (PT := T#5S);	 //simulation timer
	bInit 				: BOOL := TRUE;
	bSimulation			: BOOL := TRUE;
	bMoveToLeftReqSim 	: BOOL := TRUE;		//cmd move to left side
	bMoveToRightReqSim	: BOOL := FALSE;	//cmd move to right side
	nErrorStatus		: UINT;				//controller error output (0: no error; >0:error)
	fNoise				: LREAL;
	bNoiseUp			: BOOL;
END_VAR

iCounter := iCounter + 1;

(* initialization *)
IF bInit THEN
	A_Init();
END_IF
A_Simulation();


(* --- CYLINDER --- assign FB instance to the interface instance *)
IF NOT bEnableDiag THEN
	ipCylinder := fbCylinder;
	bDiagAvailable := FALSE;
ELSE
	ipCylinder := fbCylinderDiag;
	bDiagAvailable := FALSE;
END_IF

(* access property via interface instance *)
ipCylinder.P_TimerValue := lrTimerValue; //Set property
lrTimerValue := ipCylinder.P_TimerValue; //Get property

(* call FB via interface instance *)
bDiag := ipCylinder.M_StateMachine(
	bPosLeftReq 	:= bMoveToLeftReq,	
	bPosRightReq 	:= bMoveToRightReq,
	bAtLeftPos		=> bCylinderAtLeft,
	bAtRightPos		=> bCylinderAtRight,
);


(* --- REGULATOR --- assign FB instance to the interface instance *)
IF bEnablePID THEN
	ipRegulator := fbBasicPID;
	bPIDEnabled := TRUE;
ELSE
	ipRegulator := fbBasicP;
	bPIDEnabled := FALSE;
END_IF

(* call FB via interface instance *)
nErrorStatus := ipRegulator.M_Active(
	fSetpointValue	:= fSetpointValue,
	fActualValue	:= fActualValue,
	bReset			:= bReset,
	stRegParams		:= stRegParams,
	fCtrlOutput		=> fCtrlOutput
);

(* access property via interface instance *)
bErrorFlag := ipRegulator.P_Error; 	//Get
ipRegulator.P_Error := FALSE; 		//Set

ACTION A_Init:
bInit := FALSE;

fbCylinderDiag(tTimeOut := tTimeOutDiag);

stRegParams.fCtrlCycleTime := 0.010; 
stRegParams.fKp := 1.9; 
stRegParams.fTd := 0; 
stRegParams.fTn := 0; 
stRegParams.fTv := 0; 
fSetpointValue	:= 100;
fNoise 			:= 2.2;
bNoiseUp 		:= TRUE;
END_ACTION

ACTION A_Simulation:
Timer(IN := TRUE);

IF Timer.Q THEN
	Timer(IN := FALSE);
	IF bMoveToLeftReqSim THEN
		bMoveToLeftReqSim 	:= FALSE;
		bMoveToRightReqSim 	:= TRUE;	//cmd move to right side
 	ELSE
		bMoveToLeftReqSim 	:= TRUE;	//cmd move to left side
		bMoveToRightReqSim	:= FALSE;
	END_IF
END_IF

IF bSimulation THEN
	MEMCPY(ADR(bMoveToLeftReq), ADR(bMoveToLeftReqSim), SIZEOF(bMoveToLeftReq));
	MEMCPY(ADR(bMoveToRightReq), ADR(bMoveToRightReqSim), SIZEOF(bMoveToRightReq));

	IF fNoise >= 10 THEN
		bNoiseUp := FALSE;
	ELSIF fNoise <= -10 THEN
		bNoiseUp := TRUE;
	END_IF

	IF bNoiseUp THEN
		fNoise := fNoise + 0.01;
	ELSE
		fNoise := fNoise - 0.01;
	END_IF
	fNoise := LIMIT(-11.0, fNoise, 11.0);
  
	fActualValue := fActualValue + LIMIT(-100,fCtrlOutput,100) + fNoise;
END_IF
END_ACTION

END_FUNCTION_BLOCK

// ---- POUs/Sample OOP/Cylinder/FB_Cylinder.TcPOU
FUNCTION_BLOCK FB_Cylinder IMPLEMENTS ICylinder //regular FB that additionally implements an interface "ICylinder"
VAR_INPUT
END_VAR
VAR_OUTPUT
END_VAR
VAR
	//internal TIME variable that is being accessed via property "P_Timervalue" (Get/Set)
	tTimerValue 	: TIME := T#500MS;

	iState			: INT;
	bAtLeftPosFbk	: BOOL;
	bAtRightPosFbk	: BOOL;
	TimerReach 		: TON;
	TimerStart 		: TON;
END_VAR

;

METHOD M_StateMachine : BOOL
VAR_INPUT
	bPosLeftReq	: BOOL;
	bPosRightReq: BOOL;
END_VAR
VAR_OUTPUT
	bAtLeftPos	: BOOL;
	bAtRightPos	: BOOL;
END_VAR
// variables of a method are temporary and therefore cleared in teh next cycle 
// variables of the FB can be used for keeping variable values over many PLC cycles
(* simple cylinder with feedback  *)
CASE iState OF
0: (* at left pos *)
	bAtLeftPosFbk := TRUE;
	bAtRightPosFbk := FALSE;
	
	IF bPosRightReq THEN
		TimerStart(IN := FALSE);
		TimerReach(IN := FALSE);
		iState := iState + 1;
	END_IF

1: (* start motion to right side *)
	 TimerStart(IN := TRUE, PT := tTimerValue);
	 IF TimerStart.Q THEN
		bAtLeftPosFbk := FALSE;
		TimerStart(IN := FALSE);
		TimerReach(IN := TRUE);
		iState := iState + 1;
	 END_IF

2: (* moving *)
	 TimerReach(IN := TRUE, PT := tTimerValue);
	 IF TimerReach.Q THEN
		bAtRightPosFbk := TRUE;
		TimerReach(IN := FALSE);
		iState := iState + 1;
	 END_IF

3: (* right pos reached *)
	bAtLeftPosFbk := FALSE;
	bAtRightPosFbk := TRUE;
	
	IF bPosLeftReq THEN
		TimerStart(IN := FALSE);
		TimerReach(IN := FALSE);
		iState := iState + 1;
	END_IF

4: (* start motion to left side *)
	 TimerStart(IN := TRUE, PT := tTimerValue);
	 IF TimerStart.Q THEN
		bAtRightPosFbk := FALSE;
		TimerStart(IN := FALSE);
		TimerReach(IN := TRUE);
		iState := iState + 1;
	 END_IF

5: (* moving *)
	 TimerReach(IN := TRUE, PT := tTimerValue);
	 IF TimerReach.Q THEN
		bAtLeftPosFbk := TRUE;
		TimerReach(IN := FALSE);
		iState := 0;
	 END_IF
END_CASE

bAtLeftPos 		:= bAtLeftPosFbk;
bAtRightPos 	:= bAtRightPosFbk;

M_StateMachine 	:= FALSE;
END_METHOD

PROPERTY P_TimerValue : LREAL //encapsulates internal variable tTimerValue
GET
//read property (returns value of of internal variable)
P_TimerValue := TIME_TO_LREAL(tTimerValue) * LREAL#0.001; //convert ms (TIME) to s (LREAL)
END_GET
SET
//write property (set value of of internal variable)
tTimerValue := LREAL_TO_TIME(P_TimerValue * LREAL#1000); //convert s (LREAL) to ms (TIME)
END_SET
END_PROPERTY

END_FUNCTION_BLOCK

// ---- POUs/Sample OOP/Cylinder/FB_CylinderDiag.TcPOU
FUNCTION_BLOCK FB_CylinderDiag EXTENDS FB_Cylinder
VAR_INPUT
	tTimeOut 	  : TIME;
END_VAR
VAR
	WatchDogTimer : TON;
END_VAR

;

METHOD M_Diag : BOOL
VAR_INPUT
END_VAR
IF (iState = 0) OR (iState = 3) THEN
	WatchDogTimer(IN := FALSE, PT := tTimeOut);
ELSE
	WatchDogTimer(IN := TRUE, PT := tTimeOut);
END_IF

M_Diag := WatchDogTimer.Q;
END_METHOD

METHOD M_StateMachine : BOOL
VAR_INPUT
	bPosLeftReq  : BOOL;
	bPosRightReq : BOOL;
END_VAR
VAR_OUTPUT
	bAtLeftPos  : BOOL;
	bAtRightPos : BOOL; 
END_VAR
//call M_StateMachine of base class (FB_Cylinder) via 'SUPER^.' (access to things of FB_CylinderDiag via 'THIS^.')  
SUPER^.M_StateMachine(
	bPosLeftReq 	:= bPosLeftReq,	
	bPosRightReq 	:= bPosRightReq,
	bAtLeftPos		=> bAtLeftPos,
	bAtRightPos		=> bAtRightPos,
);

//additional diagnosis
M_StateMachine 		:= M_Diag();
END_METHOD

END_FUNCTION_BLOCK

// ---- POUs/Sample OOP/Regulator/FB_BasicP.TcPOU
FUNCTION_BLOCK FB_BasicP IMPLEMENTS IRegulator //regular FB that additionally implements an interface "IRegulator" as P-Controller
VAR CONSTANT
	nERR_NOERROR			: UINT := 0;	// no error
	nERR_INVALIDPARAM		: UINT := 1;	// invalid parameter
	nERR_INVALIDCYCLETIME	: UINT := 2;	// invalid cycle time				
END_VAR
VAR
	(* STATIC VARIABLE *)
	(* Internal Variable *)
	fE						: LREAL := 0.0;	// error input
	fE_1					: LREAL := 0.0;	// error input z^(-1)
	fY						: LREAL := 0.0;	// control output
	fY_1					: LREAL := 0.0;	// control output  z^(-1)
	fYP						: LREAL := 0.0;	// P-part
	nErrorStatus			: UINT;			// controller error output (0: no error; >0:error)
	(* Internal Parameter *)
	bInit					: BOOL	:= TRUE;// initialization flag for first cycle
	fCtrlCycleTimeOld		: LREAL	:= 0.0;
	fKpOld					: LREAL	:= 0.0;
END_VAR

;

METHOD M_Active 	: UINT
VAR_INPUT
	(* controller input  *)
	fSetpointValue	: LREAL;		// setpoint value
	fActualValue	: LREAL;		// actual value
	bReset			: BOOL;			// reset flag
	(* controller values *)
	stRegParams		: ST_RegParams;
END_VAR
VAR_OUTPUT
	fCtrlOutput		: LREAL;		// controller output command
END_VAR
(* init necessary? *)
IF (stRegParams.fCtrlCycleTime <> fCtrlCycleTimeOld) OR (stRegParams.fKp <> fKpOld) THEN
	bInit := TRUE;
END_IF

(* controller init *)
IF bInit OR bReset THEN
	(* reset internal and external variables *)
	fE	:= fE_1		:= 0.0;
	fY	:= fY_1		:= 0.0;
	fYP	:= 0.0;
	fCtrlOutput		:= 0.0;
	nErrorStatus	:= nERR_NOERROR;

	(* check cycle time parameter: (CycleTime > 0 AND CycleTme <= 60) *)
	IF ( stRegParams.fCtrlCycleTime <= 0) THEN
		nErrorStatus := nERR_INVALIDCYCLETIME;
		M_Active := nErrorStatus;
		RETURN;
	END_IF;

	(* reset *)
	IF bReset THEN
		M_Active := nErrorStatus;
		RETURN;
	END_IF

	(* set internal init flag *)
	fCtrlCycleTimeOld 	:= stRegParams.fCtrlCycleTime;
	fKpOld 				:= stRegParams.fKp;
	bInit				:= FALSE;
END_IF;

(* 3. save old variable *)
fE_1		:= fE;
fY_1		:= fY;

(* 4. set error/deviation input *)
fE	:= fSetpointValue - fActualValue;

(* 5. YP-part *)
fYp		:= stRegParams.fKp * fE;

(* 8. Ysum = YP *)
fY	:= fYP;

(* 10. set controller output *)
fCtrlOutput := fY;

M_Active := nErrorStatus;
END_METHOD

PROPERTY P_Error : BOOL
GET
P_Error := (nErrorStatus <> 0); // get error status
END_GET
SET
nErrorStatus := 0; // clear error status
END_SET
END_PROPERTY

END_FUNCTION_BLOCK

// ---- POUs/Sample OOP/Regulator/FB_BasicPID.TcPOU
FUNCTION_BLOCK FB_BasicPID IMPLEMENTS IRegulator //regular FB that additionally implements an interface "IRegulator" as PID-Controller
VAR CONSTANT
	nERR_NOERROR			: UINT := 0;	// no error
	nERR_INVALIDPARAM		: UINT := 1;	// invalid parameter
	nERR_INVALIDCYCLETIME	: UINT := 2;	// invalid cycle time				
END_VAR
VAR
	(*
		                       1               Tv * s						
	  	G(s) = Kp * ( 1 + ------------ + --------------- )				
	                         Tn * s       1 + Td * s					
	*)

	(* STATIC VARIABLE *)
	(* Internal Variable *)
	fE						: LREAL := 0.0;	// error input
	fE_1					: LREAL := 0.0;	// error input z^(-1)
	fY						: LREAL := 0.0;	// control output
	fY_1					: LREAL := 0.0;	// control output  z^(-1)
	fYP						: LREAL := 0.0;	// P-part
	fYI						: LREAL := 0.0;	// I-part			
	fYI_1					: LREAL := 0.0;	// I-part  z^(-1)	
	fYD						: LREAL := 0.0;	// D-T1-part		
	fYD_1					: LREAL := 0.0;	// D-T1-part  z^(-1)
	nErrorStatus			: UINT;			// controller error output (0: no error; >0:error)
	(* Internal Parameter *)
	bInit					: BOOL	:= TRUE;// initialization flag for first cycle
	bIsIPart				: BOOL	:= FALSE;// I-part active ?
	bIsDPart				: BOOL	:= FALSE;// D-part active ?
	fDi						: LREAL	:= 0.0;	// internal I param
	fDd						: LREAL	:= 0.0;	// internal D param
	fCd						: LREAL	:= 0.0;	// internal D param
	fCtrlCycleTimeOld		: LREAL	:= 0.0;
	fKpOld					: LREAL	:= 0.0;
	fTnOld					: LREAL	:= 0.0;
	fTvOld					: LREAL	:= 0.0;
	fTdOld					: LREAL	:= 0.0;
END_VAR

;

METHOD M_Active 	: UINT
VAR_INPUT
	(* controller input  *)
	fSetpointValue	: LREAL;		// setpoint value
	fActualValue	: LREAL;		// actual value
	bReset			: BOOL;			// reset flag
	(* controller values *)
	stRegParams		: ST_RegParams;
END_VAR
VAR_OUTPUT
	fCtrlOutput		: LREAL;		// controller output command
END_VAR
(* init necessary? *)
IF (stRegParams.fCtrlCycleTime <> fCtrlCycleTimeOld) OR (stRegParams.fKp <> fKpOld) OR (stRegParams.fTn <> fTnOld) 
	OR (stRegParams.fTv <> fTvOld) OR (stRegParams.fTd <> fTdOld) THEN
	
	bInit := TRUE;
END_IF

(* controller init *)
IF bInit OR bReset THEN
	(* reset internal and external variables *)
	fE	:= fE_1		:= 0.0;
	fY	:= fY_1		:= 0.0;
	fYP	:= 0.0;
	fYI	:= fYI_1	:= 0.0;
	fYD	:= fYD_1	:= 0.0;
	fCtrlOutput		:= 0.0;
	bIsIPart		:= FALSE;
	bIsDPart		:= FALSE;
	fCtrlOutput		:= 0.0;
	nErrorStatus	:= nERR_NOERROR;

	(* check cycle time parameter: (CycleTime > 0 AND CycleTme <= 60) *)
	IF ( stRegParams.fCtrlCycleTime <= 0) 	THEN
		nErrorStatus := nERR_INVALIDCYCLETIME;
		M_Active := nErrorStatus;
		RETURN;
	END_IF;

	(* check controller parameters: (Tn, Tv, Td >= 0) *)
	IF ( (stRegParams.fTn < 0) OR (stRegParams.fTv < 0) OR (stRegParams.fTd < 0) ) THEN
		nErrorStatus := nERR_INVALIDPARAM;
		M_Active := nErrorStatus;
		RETURN;
	END_IF;

	(* I-part *)
	IF( stRegParams.fTn > 0.0 ) THEN
		fDi := (stRegParams.fKp * stRegParams.fCtrlCycleTime) / (2.0 * stRegParams.fTn);
		bIsIPart := TRUE;
	ELSE
		fDi := 0.0;
		bIsIPart := FALSE;
	END_IF;

	(* D-part *)
	IF( stRegParams.fTv > 0.0 ) AND (stRegParams.fTd > 0.0) THEN
		fDd := (stRegParams.fKp * stRegParams.fTv) / (stRegParams.fTd + stRegParams.fCtrlCycleTime / 2.0);
		fCd := (stRegParams.fTd - stRegParams.fCtrlCycleTime / 2.0) / (stRegParams.fTd + stRegParams.fCtrlCycleTime / 2.0);
		bIsDPart := TRUE;
	ELSE
		fDd := 0.0;
		fCd := 0.0;
		bIsDPart := FALSE;
	END_IF;

	(* reset *)
	IF bReset THEN
		M_Active := nErrorStatus;
		RETURN;
	END_IF

	(* set internal init flag *)
	fCtrlCycleTimeOld 	:= stRegParams.fCtrlCycleTime;
	fKpOld 				:= stRegParams.fKp;
	fTnOld 				:= stRegParams.fTn;
	fTvOld 				:= stRegParams.fTv;
	fTdOld 				:= stRegParams.fTd;
	bInit				:= FALSE;
END_IF;

(* 3. save old variable *)
fE_1	:= fE;
fY_1	:= fY;
fYI_1	:= fYI;
fYD_1	:= fYD;

(* 4. set error/deviation input *)
fE		:= fSetpointValue - fActualValue;

(* 5. YP-part *)
fYp		:= stRegParams.fKp * fE;

(* 6. YI-part *)
IF bIsIPart THEN
	fYI := fYI_1 + fDi * (fE + fE_1);
ELSE
	fYI	:= 0.0;
END_IF;

(* 7. YD-part *)
IF bIsDPart THEN
	fYD	:=  fCd * fYD_1 + fDd * (fE - fE_1);
ELSE
	fYD	:= 0.0;
END_IF;

(* 8. Ysum = YP + YI + YD *)
fY	:= fYP + fYI + fYD;

(* 10. set controller output *)
fCtrlOutput := fY;

M_Active := nErrorStatus;
END_METHOD

PROPERTY P_Error : BOOL
GET
P_Error := (nErrorStatus <> 0); // get error status
END_GET
SET
nErrorStatus := 0; // clear error status
END_SET
END_PROPERTY

END_FUNCTION_BLOCK

// ---- POUs/Sample OOP Conveyor/FB_OOPConveyor.TcPOU
FUNCTION_BLOCK FB_OOPConveyor
VAR_INPUT
	eSampleModeIn		: E_SampleMode;	
END_VAR
VAR_IN_OUT
	AxisRef				: ARRAY [1..iMAX_AXES_REF] OF AXIS_REF;			// axis reference (process data plc/nc)
END_VAR
VAR_OUTPUT
	eSampleModeOut		: E_SampleMode;	
END_VAR
VAR
	iCounter 			: DINT;	

	//axes FB instances
	fbConv1Axis			: FB_AxisNc;
	fbConv2Axis 		: FB_VeryBasicMotor;
	fbConv3Axis 		: FB_AX5000;
	
	//axes interfaces	
	ipConv1Axis 		: I_Axis;
	ipConv2Axis 		: I_Axis;
	ipConv3Axis 		: I_Axis;
	
	//drive references
	stConv3DriveRef 	: ST_DRIVEREF;
	
	//station
	fbStation			: FB_Station;
	fbTransfer1 		: FB_TransferStation;
	fbTransfer2 		: FB_TransferStation;
	
	//conveyor
	fbInfeedConveyor 	: FB_Conveyor;
	fbConveyor2 		: FB_Conveyor;
	fbConveyor3 		: FB_Conveyor;

	//other variables
	bAllowJog			: BOOL;
	bEnableAxis1		: BOOL := TRUE;
	bJogActive			: BOOL;
	eMachineState		: E_Modes := E_SwitchingToAuto;
	iInfeedManualRequest: UDINT;
	bJogBwd AT %I*		: BOOL;
	bJogFwd AT %I*		: BOOL;
	I					: INT;
	fJogSpeed			: LREAL :=200;
	fConveyorCmdSpeed	: LREAL :=10;
	bRunConveyor		: BOOL := TRUE;
	iAnalogValue		: INT;
	bPartPresent		: BOOL;
	iAcceptPartStatus	: UDINT;
	bPickPart			: BOOL;
	iTransferPartStatus	: UDINT;
	fbTrigNewPart		: R_TRIG;
	iTransferPlacePartStatus: UDINT;
	bPlacePart			: BOOL;
	iTransfer2Status	: UDINT;
	bPickPart2			: BOOL;
	bPlacePart2			: BOOL;
	iRemoveFromConveyor3Status: UDINT;
	stOutfeedpart 		: ST_PartData;
	bRemovePart			: BOOL;
	bPartRemoved		: BOOL;
	stEmptyPart			: ST_PartData;
	bBusy				: BOOL;
	Timer				: TON := (PT := T#30s);
END_VAR

iCounter := iCounter + 1;

IF (eSampleModeIn = eSMode_OOPConv_Req) OR (eSampleModeOut = eSMode_OOPConv_Act) THEN
	//call conveyor axes
	fbConv1Axis(stAxisRef := AxisRef[1]); //FB_Axis
	fbConv2Axis(iAnalogInput := iAnalogValue, fScalingFactor:= 1, iAnalogOutput=>iAnalogValue ); //FB_VeryBasicMotor
	fbConv3Axis(stAxisRef := AxisRef[2], stDriveRef:= stConv3DriveRef); //FB_AX5000
	
	//assign axes interfaces
	ipConv1Axis := fbConv1Axis;
	ipConv2Axis := fbConv2Axis;
	ipConv3Axis := fbConv3Axis;
	
	//call conveyor FBs
	fbInfeedConveyor(fbAxis:= ipConv1Axis);
	fbConveyor2(fbAxis := ipConv2Axis);
	fbConveyor3(fbAxis := ipConv3Axis);
	
	//call stations 
	fbTransfer1(fbConveyorToPickFrom:= fbInfeedConveyor , fbConveyorToPlaceTo:= fbConveyor2 , fbStation:= fbStation);
	fbTransfer2(fbConveyorToPickFrom:= fbConveyor2 , fbConveyorToPlaceTo:= fbConveyor3 , fbStation:= fbStation);
	
	//call station
	fbStation();
	CASE eMachineState OF
		E_Disabled: 
			//Machine is disabled
			fbInfeedConveyor.P_DeviceID :=1;
			fbTransfer1.P_DeviceID := 2;
			fbStation.P_DeviceID:= 3;
			fbConveyor2.P_DeviceID := 4;
			fbConveyor3.P_DeviceID := 5;
			fbInfeedConveyor.P_MinimumSpacing := 50;
			fbInfeedConveyor.P_StartLocation := 10;
			fbInfeedConveyor.P_PickLocation := 300;
			fbConveyor2.P_MinimumSpacing:= 75;
			fbConveyor2.P_StartLocation := 10;
			fbConveyor2.P_PickLocation := 200;
			fbConveyor3.P_MinimumSpacing:= 20;
			fbConveyor3.P_StartLocation := 10;
			fbConveyor3.P_PickLocation := 600;
			FOR I := 1 TO 100 DO   
				arrParts[I].fLength := 10;
			END_FOR  
			
		E_Error: 
			;  //Machine is in an error state
			
		E_SwitchingToAuto: 
			//Reqeuest Auto from all devices 
			fbInfeedConveyor.M_Auto(bRequestAutoMode:= TRUE);
			fbStation.M_Auto(bRequestAutoMode:=TRUE );
			fbConveyor2.M_Auto(bRequestAutoMode:= TRUE);
			fbConveyor3.M_Auto(bRequestAutoMode:= TRUE);
			fbTransfer1.M_Auto(bRequestAutoMode:= TRUE);
			
			// If all devices are in auto mode then the machine is in Auto mode
			IF fbInfeedConveyor.P_CurrentState = E_Auto  
			  AND fbStation.P_CurrentState = E_Auto 
			  AND fbConveyor2.P_CurrentState = E_Auto 
			  AND fbTransfer1.P_CurrentState = E_Auto
			  AND fbConveyor3.P_CurrentState = E_Auto THEN 
					eMachineState:= E_Auto;
					fbInfeedConveyor.M_Auto(bRequestAutoMode:= FALSE);
					fbTransfer1.M_Auto(bRequestAutoMode := FALSE);
					fbStation.M_Auto(bRequestAutoMode:=FALSE);
					fbConveyor2.M_Auto(bRequestAutoMode:= FALSE);
					fbConveyor3.M_Auto(bRequestAutoMode:= FALSE);
					
			//If any devices are in Error mode then the machine is in the error state
			ELSIF fbInfeedConveyor.P_CurrentState = E_Error  
			  OR fbStation.P_CurrentState = E_Error 
			  OR fbConveyor2.P_CurrentState = E_Error     
			  OR fbTransfer1.P_CurrentState = E_Error
			  OR fbConveyor3.P_CurrentState = E_Error THEN  
					eMachineState:= E_Error;
					fbTransfer1.M_Auto(bRequestAutoMode := FALSE);
					fbInfeedConveyor.M_Auto(bRequestAutoMode:= FALSE);
					fbStation.M_Auto(bRequestAutoMode:=FALSE );
					fbConveyor2.M_Auto(bRequestAutoMode:= FALSE);
					fbConveyor3.M_Auto(bRequestAutoMode:= FALSE);
			END_IF
			
		E_SwitchingToManual:
			//Reqeuest Manual from all devices 
			fbInfeedConveyor.M_Manual(bRequestManualMode:= TRUE);
			fbStation.M_Manual(bRequestManualMode:= TRUE);
			fbConveyor2.M_Manual(bRequestManualMode:=TRUE );
			fbConveyor3.M_Manual(bRequestManualMode:=TRUE );
			fbTransfer1.M_Manual(bRequestManualMode:=TRUE);
			// If all devices are in Manual mode then the machine is in Manual mode
			IF fbInfeedConveyor.P_CurrentState = E_Manual 
			  AND fbConveyor2.P_CurrentState = E_Manual 
			  AND fbConveyor3.P_CurrentState = E_Manual
			  AND fbTransfer1.P_CurrentState = E_Manual
			  AND fbStation.P_CurrentState = E_Manual  THEN
					eMachineState:= E_Manual;
					fbInfeedConveyor.M_Manual(bRequestManualMode:= FALSE);
					fbStation.M_Manual(bRequestManualMode:= FALSE);
					fbConveyor2.M_Manual(bRequestManualMode:=FALSE );
					fbTransfer1.M_Manual(bRequestManualMode:=FALSE);
					fbConveyor3.M_Manual(bRequestManualMode:=FALSE);
			//If any devices are in Error mode then the machine is in the error state
			ELSIF fbInfeedConveyor.P_CurrentState = E_Error 
			  OR fbConveyor2.P_CurrentState = E_Error 
			  OR fbConveyor3.P_CurrentState = E_Error
			  OR fbTransfer1.P_CurrentState = E_Error
			  OR  fbStation.P_CurrentState = E_Error THEN 
					eMachineState:= E_Error;
					fbInfeedConveyor.M_Manual(bRequestManualMode:= FALSE);
					fbStation.M_Manual(bRequestManualMode:= FALSE);
					fbTransfer1.M_Manual(bRequestManualMode:=FALSE);
					fbConveyor2.M_Manual(bRequestManualMode:=FALSE );
					fbConveyor3.M_Manual(bRequestManualMode:=FALSE);
			END_IF
		
		E_Resetting: 
			fbInfeedConveyor.M_Reset(bRequestReset:=TRUE );
			fbConveyor2.M_Reset(bRequestReset:=TRUE);
			fbConveyor3.M_Reset(bRequestReset:=TRUE);
			fbStation.M_Reset(bRequestReset:= TRUE);
			IF fbInfeedConveyor.P_CurrentState = E_Reset 
			  AND fbConveyor2.P_CurrentState = E_Reset 
			  AND fbConveyor3.P_CurrentState = E_Reset
			  AND fbStation.P_CurrentState = E_Reset THEN
				eMachineState := E_Reset;
				fbInfeedConveyor.M_Reset(bRequestReset:=FALSE );
				fbConveyor2.M_Reset(bRequestReset:=FALSE);
				fbConveyor3.M_Reset(bRequestReset:=FALSE);
				fbStation.M_Reset(bRequestReset:= FALSE);
			ELSIF fbInfeedConveyor.P_CurrentState = E_Error   
			  OR fbConveyor2.P_CurrentState = E_Error 
			  OR fbConveyor3.P_CurrentState = E_Error
			  OR  fbStation.P_CurrentState = E_Error THEN 
					eMachineState:= E_Error;
					fbInfeedConveyor.M_Reset(bRequestReset:=FALSE );
					fbConveyor2.M_Reset(bRequestReset:=FALSE);
					fbConveyor3.M_Reset(bRequestReset:=FALSE);
					fbStation.M_Reset(bRequestReset:= FALSE);
			END_IF
		
		E_Reset: 
			// Machine has been reset and awaits a mode change to Manual or Auto
			 ;
	
							
		E_Manual :  
			// Manual Mode allow all manual commands
			fbInfeedConveyor.bJogConveyorFwd:=bJogFwd; 
			fbInfeedConveyor.bJogConveyorBwd:=bJogBwd; 
			fbInfeedConveyor.fJogSpeed:= fJogSpeed;
			fbConveyor2.fJogSpeed:=fJogSpeed;
			fbConveyor2.bJogConveyorFwd:=bJogFwd; 
			fbConveyor2.bJogConveyorBwd:=bJogBwd;
			fbConveyor3.bJogConveyorFwd:=bJogFwd;
			fbConveyor3.bJogConveyorBwd:=bJogBwd; 
			fbConveyor3.fJogSpeed:=fJogSpeed;
			
		E_Auto :		
			fbInfeedConveyor.fCmdSpeed:= fConveyorCmdSpeed;
			fbInfeedConveyor.bRunConveyor := bRunConveyor;
			fbConveyor2.bRunConveyor := bRunConveyor;
			fbConveyor2.fCmdSpeed := fConveyorCmdSpeed +5;
			fbConveyor3.bRunConveyor := bRunConveyor;
			fbConveyor3.fCmdSpeed := fConveyorCmdSpeed +3;
			//button triggers a part is presetn
			fbTrigNewPart(CLK:= bPartPresent);
			IF fbTrigNewPart.Q THEN 
				arrParts[1].iIDNumber:= arrParts[1].iIDNumber + 5 ;
			END_IF
			iAcceptPartStatus := fbInfeedConveyor.M_AcceptPart(bPartPresentAtEntrance:=bPartPresent , stPartAtEntrance:=arrParts[1] );
			//Part has been accepted by conveyor 
			IF iAcceptPartStatus = 3 THEN 
				bPartPresent := FALSE;
			END_IF
			iTransferPartStatus := fbTransfer1.M_PickPart(bGetPart:=bPickPart, bPartAvailable := fbInfeedConveyor.bPartInPickLocation );
			IF  bPlacePart (*fbTransfer1.bHavePart*) THEN 
				iTransferPlacePartStatus := fbTransfer1.M_PlacePart(bPlacePart:=TRUE );
			END_IF
			iTransfer2Status := fbTransfer2.M_PickPart(bGetPart:=bPickPart2, bPartAvailable := fbConveyor2.bPartInPickLocation );
			IF  bPlacePart2 (*fbTransfer1.bHavePart*) THEN 
				iTransfer2Status := fbTransfer2.M_PlacePart(bPlacePart:=TRUE);
			END_IF
	
			IF fbConveyor3.bPartInPickLocation THEN 
				bRemovePart := TRUE;
			END_IF
			IF stOutfeedpart.iIDNumber <>0 THEN 
				bPartRemoved := TRUE; 
			END_IF 	
			iRemoveFromConveyor3Status := fbConveyor3.M_ReleasePart(bReleasePartReq:=bRemovePart , bPartHandedOff:=bPartRemoved , stPartToRelease=>stOutfeedpart );
			IF iRemoveFromConveyor3Status = 3 THEN 
				stOutfeedpart := stEmptyPart;
				bRemovePart:=FALSE;
				bPartRemoved := FALSE;
			END_IF	
			
	END_CASE

	Timer(IN := TRUE);
	IF Timer.Q THEN
		Timer(IN := FALSE);
		bBusy := FALSE;
	ELSE
		bBusy := TRUE;
	END_IF
	
	IF bBusy THEN
		eSampleModeOut := eSMode_OOPConv_Act;
	ELSE
		eSampleModeOut := eSMode_Idle;
	END_IF
END_IF

END_FUNCTION_BLOCK

// ---- POUs/Sample OOP Conveyor/Axis Blocks/FB_AxisNc.TcPOU
FUNCTION_BLOCK FB_AxisNc IMPLEMENTS I_Axis
VAR_INPUT
END_VAR
VAR_OUTPUT
END_VAR
VAR_IN_OUT
	stAxisRef 		: AXIS_REF;
END_VAR
VAR
//Enable	
	fbMCPower		: MC_Power;
	bEnableAxis		: BOOL;
	fbTrigEnable	: R_TRIG;
	
//Jog	
	fbJog			: MC_Jog;
	bJogAxisFwd		: BOOL;
	bJogAxisBwd		: BOOL;
	fJogAxisSpeed	: LREAL;
	fbJogErrTrig	: R_TRIG;
	bJogError		: BOOL;
	udiJogErrID		: UDINT;
	
//Move Velocity 	
	fbMoveVelocity 	: MC_MoveVelocity;
	eAxisDirection	: MC_Direction;
	fbStartMoveVelocity: R_TRIG;
	iVeloMoveSeq	: INT;
	
//Reset	
	fbMCReset		: MC_Reset;
	fbTrigResetSeq	: R_TRIG;
	iResetSeq		: INT;
	bError			: BOOL;
	udiErrorID		: UDINT;
	fbTrigStop		: R_TRIG;
	iStopSeq		: INT;
	fbMCStop		: MC_Stop;
END_VAR

stAxisRef.ReadStatus();

//the MC_Power block is one that should be called every cycle to allow for a very quick disabling of the axis
fbMCPower(
	Enable			:= bEnableAxis , 
	Enable_Positive	:= bEnableAxis , 
	Enable_Negative	:= bEnableAxis , 
	Override		:= 100.0 , 
	Axis			:= stAxisRef );

METHOD M_Disable : UDINT
VAR_INPUT
	bDisable : BOOL;
END_VAR
//The result of the method is an unsigned double integer
// 0 = idle 
// 1 = busy
// 3 = complete
// Any other number = Error
IF NOT bDisable THEN
	M_Disable := 0;
END_IF

IF bDisable THEN 
	bEnableAxis := FALSE;
	M_Disable := 1;
END_IF

IF NOT fbMCPower.Status THEN
	M_Disable := 3;
END_IF
END_METHOD

METHOD M_Enable : UDINT
VAR_INPUT
	bEnable : BOOL;
END_VAR
//The result of the method is an unsigned double integer
// 0 = idle 
// 1 = busy
// 3 = complete
// Any other number = Error
IF bEnable THEN
	bEnableAxis := TRUE;
	M_Enable := 1;
END_IF

IF fbMCPower.Status THEN
	M_Enable := 3;
END_IF

IF fbMCPower.Error THEN
	M_Enable :=fbMCPower.ErrorID;
END_IF

IF NOT bEnable THEN
	M_Enable := 0;
END_IF
END_METHOD

METHOD M_HardwareReset : UDINT
VAR_INPUT
	bReset	: BOOL;
END_VAR
//The result of the method is an unsigned double integer
// 0 = idle 
// 1 = busy
// 3 = complete
// Any other number = Error
// Default result for the method is that it completes
IF bReset THEN
	M_HardwareReset := 3;
END_IF

IF NOT bReset THEN
	M_HardwareReset := 0;
END_IF
END_METHOD

METHOD M_Jog : UDINT
VAR_INPUT
	bJogFwd 	: BOOL;
	bJogBwd 	: BOOL;
	fJogSpeed 	: LREAL;
END_VAR
//The result of the method is an unsigned double integer
// 0 = idle 
// 1 = busy
// 3 = complete
// Any other number = Error
IF bJogFwd AND NOT bJogBwd THEN
	bJogAxisFwd := TRUE;
	bJogAxisBwd := FALSE;
ELSIF bJogBwd AND NOT bJogFwd THEN
	bJogAxisBwd := TRUE;
	bJogAxisFwd := FALSE;
ELSE
	bJogAxisBwd := FALSE;
	bJogAxisFwd := FALSE;
END_IF

fbJog(
	JogForward	:= bJogAxisFwd, 
	JogBackwards:= bJogAxisBwd, 
	Velocity	:= fJogSpeed, 
	Mode 		:= MC_JOGMODE_CONTINOUS,
	Axis		:= stAxisRef
);
	
fbJogErrTrig(CLK := fbJog.Error);
IF fbJogErrTrig.Q THEN
	bJogError:=TRUE;
	udiJogErrID := fbJog.ErrorID;
END_IF

IF fbJog.Active THEN
	M_Jog := 1;
ELSIF fbJog.Error THEN
	M_Jog := fbJog.ErrorID;
ELSE
	M_Jog := 0;
END_IF
END_METHOD

METHOD M_Reset : UDINT
VAR_INPUT
	bReset : BOOL;
END_VAR
//The result of the method is an unsigned double integer
// 0 = idle 
// 1 = busy
// 3 = complete
// Any other number = Error
VAR
	udiHardwareResetResult:UDINT;
END_VAR
fbTrigResetSeq(CLK:=bReset);
IF fbTrigResetSeq.Q THEN
	M_Reset		:= 1;
	iResetSeq	:= 10;
END_IF

IF NOT bReset THEN
	M_Reset 	:= 0;
END_IF

CASE iResetSeq OF 
	0: (* Idle*)
		fbMCReset(Execute := FALSE, Axis := stAxisRef);
		
	10: (*If necessary reset the hardware first*)
		M_HardwareReset(bReset:=TRUE);
		iResetSeq := 10;	
	20: 
		udiHardwareResetResult := M_HardwareReset(bReset:=TRUE);   
		IF udiHardwareResetResult = 3 THEN // Hardware reset successful
			M_HardwareReset(bReset:=FALSE);
			iResetSeq := 30;
		ELSIF udiHardwareResetResult > 3 THEN // Hardware reset faulted
			M_Reset := udiHardwareResetResult;
			iResetSeq:= 0;			
		END_IF
		fbMCReset(Execute:=TRUE ,Axis:= stAxisRef);
		iResetSeq := 30;
	30:
		fbMCReset(Axis:=stAxisRef);
		IF fbMCReset.Done OR fbMCReset.Error THEN
			fbMCReset(Execute:=FALSE,Axis:=stAxisRef);
			iResetSeq := 0;
			IF fbMCReset.Error THEN
				M_Reset := fbMCReset.ErrorID;
			ELSE
				iResetSeq:= 0;		
				M_Reset:=2;
			END_IF
		END_IF
END_CASE
END_METHOD

METHOD M_Speed : UDINT
VAR_INPUT
	bMoveVelocity 	: BOOL;
	fSpeed 			: LREAL;
END_VAR
//The result of the method is an unsigned double integer
// 0 = idle 
// 1 = busy
// 3 = complete
// Any other number = Error
//Determine the dirction of the velocity command
IF fSpeed > 0 THEN
	eAxisDirection := MC_Positive_Direction; 
ELSE
	eAxisDirection := MC_Negative_Direction;
END_IF
//Look for a trigger 
fbStartMoveVelocity(CLK:= bMoveVelocity);
IF fbStartMoveVelocity.Q THEN 
	iVeloMoveSeq := 10;
	M_Speed:=1;
	fbMoveVelocity(Execute:= FALSE,Axis:=stAxisRef);
END_IF
// If the bMoveVelocity bit is off clear the Method
IF NOT bMoveVelocity THEN
	M_Speed := 0;
END_IF

CASE iVeloMoveSeq OF
	0: (*Idle*)
		fbMoveVelocity(Execute:=FALSE,Axis:=stAxisRef);
	10: (*Initiate Move Velocity command*)
		fbMoveVelocity(
			Execute:= TRUE , 
			Velocity:= ABS(fSpeed), 
			Direction:= eAxisDirection , 
			Axis:=stAxisRef);
		iVeloMoveSeq := 20;
		
	20: (*Wait for axis to reach velocity or error out*)
		fbMoveVelocity(Axis:=stAxisRef);
		IF fbMoveVelocity.InVelocity OR fbMoveVelocity.Error THEN
			IF fbMoveVelocity.Error THEN
				M_Speed := fbMoveVelocity.ErrorID;
			END_IF			
			fbMoveVelocity(Execute:= FALSE,Axis:=stAxisRef);
			iVeloMoveSeq:=0;
			M_Speed:=3;
		END_IF
END_CASE
END_METHOD

METHOD M_Stop : UDINT
VAR_INPUT
	bStop	: BOOL;
END_VAR
//The result of the method is an unsigned double integer
// 0 = idle 
// 1 = busy
// 3 = complete
// Any other number = Error
VAR

END_VAR
//Look for a trigger 
fbTrigStop(CLK:= bStop);
IF fbTrigStop.Q THEN 
	iStopSeq := 10;
	M_Stop:=1;
END_IF
// If the bMoveVelocity bit is off clear the Method
IF NOT bStop THEN
	M_Stop := 0;
END_IF

CASE iStopSeq OF
	0: (*Idle*)
		fbMCStop(Execute:=FALSE,Axis:=stAxisRef);
	10: (*Initiate Move Velocity command*)
		fbMCStop(Execute:= TRUE,Axis:=stAxisRef);
		iStopSeq := 20;
		
	20: (*Wait for axis to reach velocity or error out*)
		fbMCStop(Axis:=stAxisRef);
		IF fbMCStop.Done OR fbMCStop.Error THEN
			IF fbMCStop.Error THEN
				M_Stop := fbMCStop.ErrorID;
			END_IF			
			fbMCStop(Execute:= FALSE,Axis:=stAxisRef);
			iStopSeq:=0;
			M_Stop:=3;
		END_IF
END_CASE
END_METHOD

PROPERTY P_CurrentPosition : LREAL
GET
P_CurrentPosition :=  stAxisRef.NcToPlc.ActPos;
END_GET
SET
END_SET
END_PROPERTY

PROPERTY P_CurrentSpeed : LREAL
GET
P_CurrentSpeed := stAxisRef.NcToPlc.ActVelo;
END_GET
SET
// setting the current speed is not allowed
;
END_SET
END_PROPERTY

PROPERTY P_Error : BOOL
GET
//Report Errors with the most important first 
// Axis Hardware Failure
// NC Axis Failure
//Move command errors are returned by their respective method calls
P_Error := stAxisRef.Status.Error;
END_GET
SET
//Allow user to externally clear error.
IF P_Error = FALSE THEN
	udiErrorID	:= 0;
	bError 		:= FALSE;
END_IF
END_SET
END_PROPERTY

PROPERTY P_ErrorID : UDINT
GET
P_ErrorID := udiErrorID;
END_GET
SET
IF P_ErrorID = 0 THEN
	bError		:= FALSE;
	udiErrorID	:= 0;
END_IF
END_SET
END_PROPERTY

PROPERTY P_Ready : BOOL
GET
IF stAxisRef.Status.ControlLoopClosed AND NOT stAxisRef.Status.Error THEN
	P_Ready := TRUE;
ELSE
	P_Ready := FALSE;
END_IF
END_GET
SET
;
END_SET
END_PROPERTY

END_FUNCTION_BLOCK

// ---- POUs/Sample OOP Conveyor/Axis Blocks/FB_VeryBasicMotor.TcPOU
FUNCTION_BLOCK FB_VeryBasicMotor IMPLEMENTS I_Axis
VAR_INPUT
	iAnalogInput 	: INT; //Feedback from hardware
	// Scaling of feedback/command values
	fScalingFactor	: LREAL := 1;
END_VAR
VAR_OUTPUT
	iAnalogOutput 	: INT;  //Output to hardware
END_VAR
VAR
	// Disable Analog Output
	bDisableOutput	: BOOL; //Output is disabled
	bJoggingFwd		: BOOL; //Jogging Fwd
	bJoggingBwd		: BOOL; //Jogging bwd
	bMoveAtVelocity	: BOOL;  //moving at velocity
	fCurrentPosition: LREAL;
END_VAR

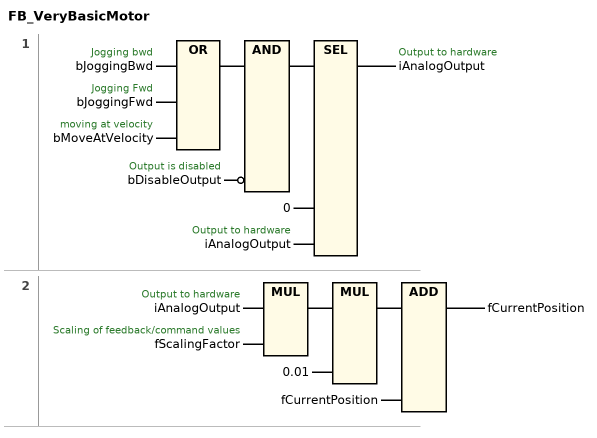
// NETWORK 1
//   bJoggingBwd: Jogging bwd
//   bJoggingFwd: Jogging Fwd
//   bMoveAtVelocity: moving at velocity
//   bDisableOutput: Output is disabled
//   iAnalogOutput: Output to hardware
iAnalogOutput := SEL((bJoggingBwd OR bJoggingFwd OR bMoveAtVelocity) AND NOT bDisableOutput, 0, iAnalogOutput);

// NETWORK 2
//   iAnalogOutput: Output to hardware
//   fScalingFactor: Scaling of feedback/command values
fCurrentPosition := (iAnalogOutput * fScalingFactor) * 0.01 + fCurrentPosition;

METHOD M_Disable : UDINT  //Result of Method
VAR_INPUT
	bDisable	: BOOL; //Input to Method
END_VAR
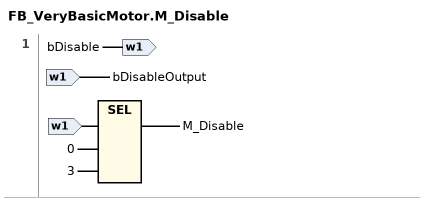
// NETWORK 1
bDisableOutput := bDisable;
M_Disable := SEL(bDisable, 0, 3);
END_METHOD

METHOD M_Enable : UDINT //Method Result
VAR_INPUT
	bEnable	: BOOL;  //Enable Output
END_VAR

VAR
	b1: BOOL;
	b2: BOOL;
END_VAR
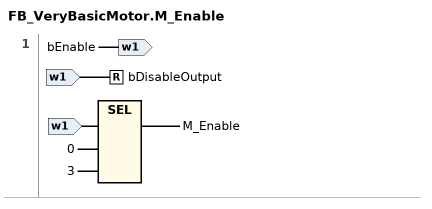
// NETWORK 1
bDisableOutput R= bEnable;
M_Enable := SEL(bEnable, 0, 3);
END_METHOD

METHOD M_HardwareReset : UDINT  //Result of Method Call
VAR_INPUT
	bReset	: BOOL;  //Bit to request hardware reset
END_VAR
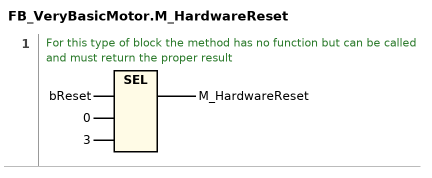
// NETWORK 1
// For this type of block the method has no function but can be called
// and must return the proper result
M_HardwareReset := SEL(bReset, 0, 3);
END_METHOD

METHOD M_Jog : UDINT //Output of block 0 idle 1 busy 3 complete
VAR_INPUT
	bJogFwd	: BOOL;  //Jog fwd command
	bJogBwd	: BOOL; // Jog bwd command
	fJogSpeed	: LREAL;  //speed to jog at
END_VAR

VAR
	
	v1 : LREAL; 
END_VAR
VAR_INST // added by the converter: edge detectors and wires of the graphical bodies
    _w1, _w2 : BOOL;
END_VAR
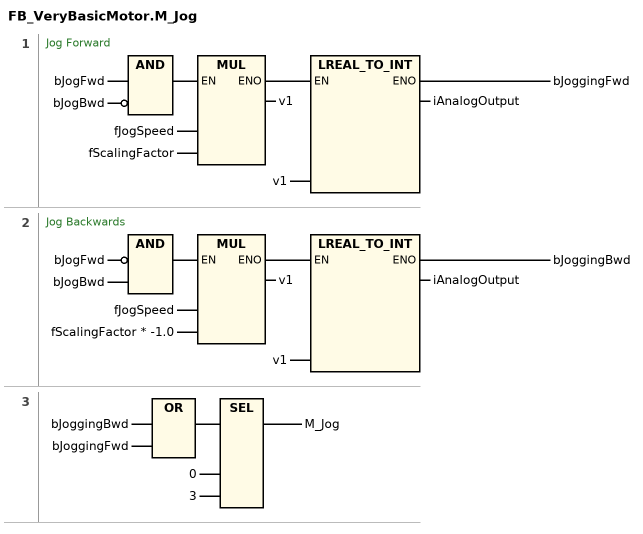
// NETWORK 1
// Jog Forward
_w1 := bJogFwd AND NOT bJogBwd;
IF _w1 THEN v1 := fJogSpeed * fScalingFactor; END_IF
IF _w1 THEN iAnalogOutput := LREAL_TO_INT(v1); END_IF
bJoggingFwd := _w1;

// NETWORK 2
// Jog Backwards
_w2 := NOT bJogFwd AND bJogBwd;
IF _w2 THEN v1 := fJogSpeed * (fScalingFactor * -1.0); END_IF
IF _w2 THEN iAnalogOutput := LREAL_TO_INT(v1); END_IF
bJoggingBwd := _w2;

// NETWORK 3
M_Jog := SEL(bJoggingBwd OR bJoggingFwd, 0, 3);
END_METHOD

METHOD M_Reset : UDINT
VAR_INPUT
	bReset	: BOOL;
END_VAR
END_METHOD

METHOD M_Speed : UDINT
VAR_INPUT
	bMoveVelocity	: BOOL;
	fSpeed	: LREAL;
END_VAR
VAR
	v1:LREAL;
END_VAR
VAR_INST // added by the converter: edge detectors and wires of the graphical bodies
    _w1 : BOOL;
END_VAR
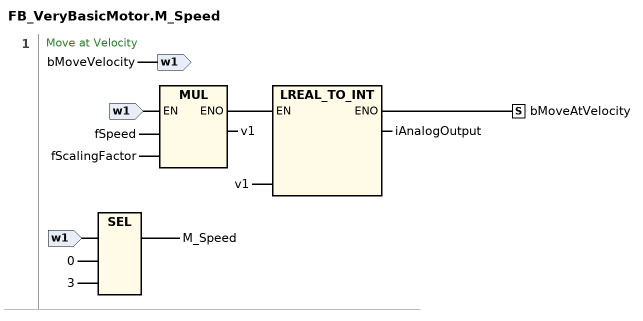
// NETWORK 1
// Move at Velocity
_w1 := bMoveVelocity;
IF _w1 THEN v1 := fSpeed * fScalingFactor; END_IF
IF _w1 THEN iAnalogOutput := LREAL_TO_INT(v1); END_IF
bMoveAtVelocity S= _w1;
M_Speed := SEL(bMoveVelocity, 0, 3);
END_METHOD

METHOD M_Stop : UDINT
VAR_INPUT
	bStop	: BOOL;
END_VAR

VAR

END_VAR
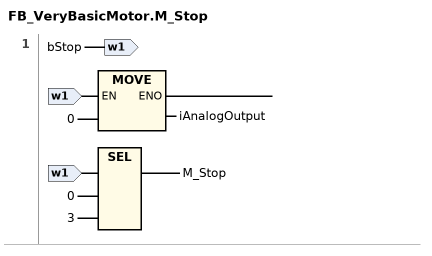
// NETWORK 1
IF bStop THEN iAnalogOutput := 0; END_IF
M_Stop := SEL(bStop, 0, 3);
END_METHOD

PROPERTY P_CurrentPosition : LREAL
GET
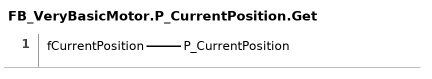
// NETWORK 1
P_CurrentPosition := fCurrentPosition;
END_GET
SET
END_SET
END_PROPERTY

PROPERTY P_CurrentSpeed : LREAL
GET
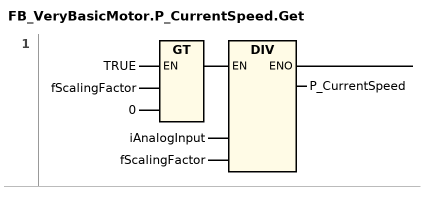
// NETWORK 1
IF fScalingFactor > 0 THEN P_CurrentSpeed := iAnalogInput / fScalingFactor; END_IF
END_GET
SET
END_SET
END_PROPERTY

PROPERTY P_Error : BOOL
GET
END_GET
SET
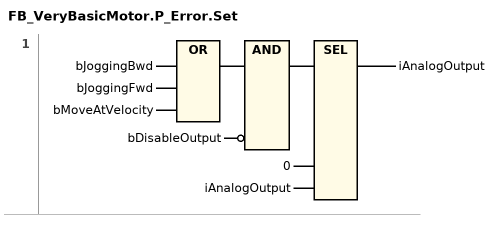
// NETWORK 1
iAnalogOutput := SEL((bJoggingBwd OR bJoggingFwd OR bMoveAtVelocity) AND NOT bDisableOutput, 0, iAnalogOutput);
END_SET
END_PROPERTY

PROPERTY P_ErrorID : UDINT
GET
END_GET
SET
END_SET
END_PROPERTY

PROPERTY P_Ready : BOOL
GET
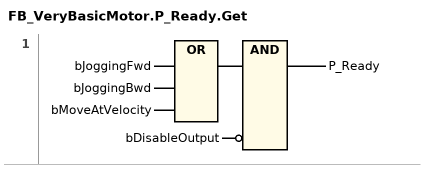
// NETWORK 1
P_Ready := (bJoggingFwd OR bJoggingBwd OR bMoveAtVelocity) AND NOT bDisableOutput;
END_GET
SET
END_SET
END_PROPERTY

END_FUNCTION_BLOCK

// ---- POUs/Sample OOP Conveyor/Axis Blocks/FB_AX5000.TcPOU
FUNCTION_BLOCK FB_AX5000 EXTENDS FB_AxisNc
VAR_INPUT
END_VAR
VAR_OUTPUT
END_VAR
VAR_IN_OUT
	stDriveRef 			: ST_DRIVEREF;
END_VAR
VAR
	//variables for the hardware reset 
	fbTrigNotBusy		: F_TRIG;
	bNotBusy			: BOOL;
	fbTrigResetNotBusy	: F_TRIG;
	fbSOEReset			: FB_SoEReset;
END_VAR

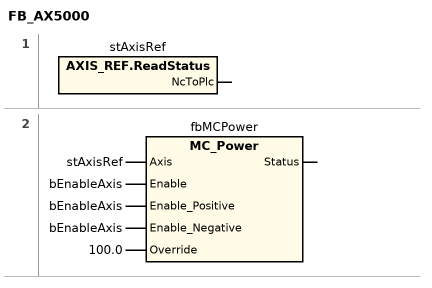
// NETWORK 1
stAxisRef.ReadStatus();

// NETWORK 2
//   fbMCPower: Enable
fbMCPower(
    Axis := stAxisRef,
    Enable := bEnableAxis,
    Enable_Positive := bEnableAxis,
    Enable_Negative := bEnableAxis,
    Override := 100.0); // MC_Power

METHOD PUBLIC M_HardwareReset : UDINT
//This method override the hardware reset method of the Inherited FB_AxisBlock
//in order to perform commands specific to resetting an AX5000 Drive
VAR_INPUT
	bReset : BOOL;
END_VAR
//Result of the Reset method is 
// 0 : Idle
// 1 : busy
// 3 : complete
// > 3 Error returned by associated function blocks
VAR
	
	
END_VAR
VAR_INST // added by the converter: edge detectors and wires of the graphical bodies
    _w1, _w2 : BOOL;
END_VAR
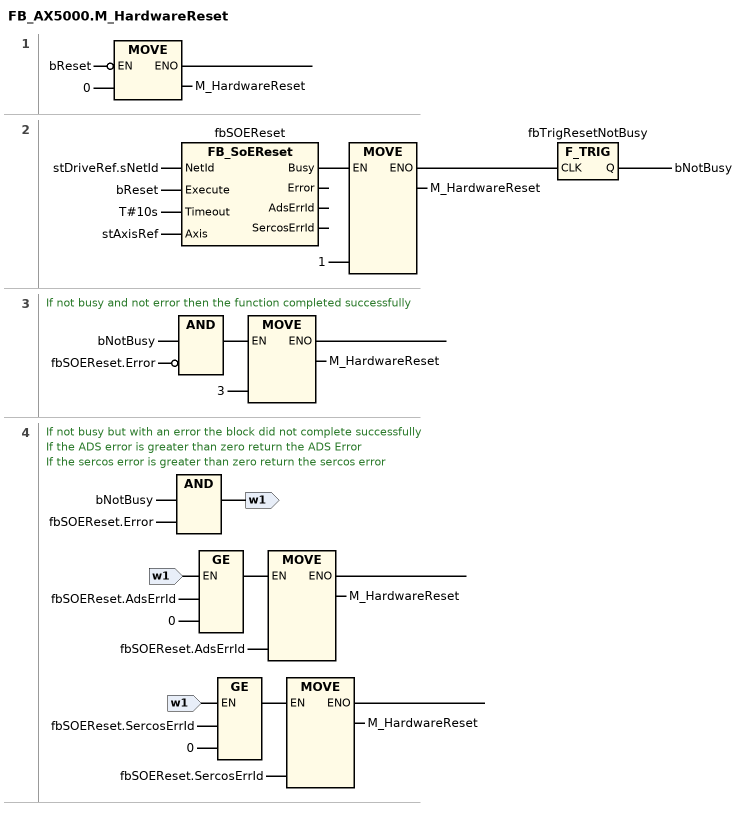
// NETWORK 1
IF NOT bReset THEN M_HardwareReset := 0; END_IF

// NETWORK 2
fbSOEReset(NetId := stDriveRef.sNetId, Execute := bReset, Timeout := T#10s, Axis := stAxisRef); // FB_SoEReset
_w1 := fbSOEReset.Busy;
IF _w1 THEN M_HardwareReset := 1; END_IF
fbTrigResetNotBusy(CLK := _w1); // F_TRIG
bNotBusy := fbTrigResetNotBusy.Q;

// NETWORK 3
// If not busy and not error then the function completed successfully
IF bNotBusy AND NOT fbSOEReset.Error THEN M_HardwareReset := 3; END_IF

// NETWORK 4
// If not busy but with an error the block did not complete successfully
// If the ADS error is greater than zero return the ADS Error
// If the sercos error is greater than zero return the sercos error
_w2 := bNotBusy AND fbSOEReset.Error;
IF _w2 AND fbSOEReset.AdsErrId >= 0 THEN M_HardwareReset := fbSOEReset.AdsErrId; END_IF
IF _w2 AND fbSOEReset.SercosErrId >= 0 THEN M_HardwareReset := fbSOEReset.SercosErrId; END_IF
END_METHOD

END_FUNCTION_BLOCK

// ---- POUs/Sample OOP Conveyor/Device And Station Blocks/FB_Station.TcPOU
FUNCTION_BLOCK FB_Station EXTENDS FB_Device
VAR_INPUT
END_VAR
VAR_OUTPUT
END_VAR
VAR
END_VAR

END_FUNCTION_BLOCK

// ---- POUs/Sample OOP Conveyor/Device And Station Blocks/FB_Device.TcPOU
FUNCTION_BLOCK FB_Device IMPLEMENTS I_Mode
VAR_INPUT
END_VAR
VAR_OUTPUT
END_VAR
VAR
	eCurrentState 	: E_Modes;
	fbTrigAutoMode	: R_TRIG;
	iSwitchAutoSeq	: INT;
	fbTrigManualMode: R_TRIG;
	iSwitchManualSeq: INT;
	iDeviceID		: UDINT;
END_VAR

P_DeviceID := iDeviceID;

METHOD M_Auto : UDINT
VAR_INPUT
	bRequestAutoMode	: BOOL;
END_VAR
// Method confirms to the user it has complteted or that it is busy
// 0: idle
// 1: busy
// 3: complete
// > 3 Error condition
fbTrigAutoMode(CLK:= bRequestAutoMode);
IF fbTrigAutoMode.Q THEN
	iSwitchAutoSeq := 10;
	M_Auto:=1;
END_IF

CASE iSwitchAutoSeq OF
	0: (*Idle*)
		;
	10: (*wait for all sub components to declare Auto state*)
		iSwitchAutoSeq := 20;
		eCurrentState:= E_SwitchingToAuto;
		M_Auto := 1;
	
	20: (*once all devices are in Auto confirm auto mode*)
		eCurrentState := E_Auto;
		iSwitchAutoSeq := 0;
		M_Auto:=3;
END_CASE
END_METHOD

METHOD M_Disable : UDINT
VAR_INPUT
	bDisable : BOOL;
END_VAR
;
END_METHOD

METHOD M_Manual : UDINT
VAR_INPUT
	bRequestManualMode	: BOOL;
END_VAR
fbTrigManualMode(CLK:= bRequestManualMode);
IF fbTrigManualMode.Q THEN
	iSwitchManualSeq := 10;
	M_Manual:=1;
END_IF

CASE iSwitchManualSeq OF
	0: (*Idle*)
		;
	10: (*wait for all sub components to declare Manual state*)
		iSwitchManualSeq := 20;
		eCurrentState:= E_SwitchingToManual;
	
	20: (*once all devices are in Manual confirm Manual mode*)
		eCurrentState := E_Manual;
		iSwitchManualSeq := 0;
		M_Manual:=3;
END_CASE
END_METHOD

METHOD M_Reset : UDINT
VAR_INPUT
	bRequestReset	: BOOL;
END_VAR

VAR
	fbTrigReset: R_TRIG;
	iResetSeq: INT;
END_VAR
fbTrigReset(CLK:= bRequestReset);
IF fbTrigReset.Q THEN
	iResetSeq := 10;
	M_Reset:=1;
END_IF

CASE iResetSeq OF
	0: (*Idle*)
		;
	10: (*wait for all sub components to declare Manual state*)
		iResetSeq := 20;
		eCurrentState:= E_Resetting;
	
	20: (*once all devices are in Manual confirm Manual mode*)
		eCurrentState := E_Reset;
		iResetSeq := 0;
		M_Reset:=3;
END_CASE
END_METHOD

PROPERTY P_CurrentState : E_Modes
GET
P_CurrentState:=eCurrentState;
END_GET
SET
//It is not allowed to set the state of the module
;
END_SET
END_PROPERTY

PROPERTY PUBLIC P_DeviceID  : UDINT
GET
P_DeviceID := iDeviceID	;
END_GET
SET
iDeviceID := P_DeviceID;
END_SET
END_PROPERTY

END_FUNCTION_BLOCK

// ---- POUs/Sample OOP Conveyor/Device And Station Blocks/FB_TransferStation.TcPOU
FUNCTION_BLOCK FB_TransferStation EXTENDS FB_Device
VAR_INPUT
END_VAR
VAR_OUTPUT
	bHavePart 				: BOOL;
END_VAR
VAR_IN_OUT
	fbConveyorToPickFrom 	: FB_Conveyor;
	fbConveyorToPlaceTo		: FB_Conveyor;
	fbStation 				: FB_Station;
END_VAR
VAR
	fbStartGetPartSeq		: R_TRIG;
	iGetPartSeq				: INT;
	stPart					: ST_PartData;
	iPlacePartSeq			: INT;
	iConveyorAcceptSeq		: UDINT;
	iConvReleasePartStatus	: UDINT;
	iConveyorAcceptStatus	: UDINT;
	fbTrigPlacePartSeq		: R_TRIG;
	stEmptyPart				: ST_PartData;
END_VAR

METHOD PUBLIC M_PickPart : UDINT
VAR_INPUT
	bGetPart : BOOL;
	bPartAvailable : BOOL;
END_VAR
VAR_OUTPUT 

END_VAR
VAR
	
END_VAR
fbStartGetPartSeq(CLK:=bGetPart AND NOT bHavePart AND bPartAvailable);
IF fbStartGetPartSeq.Q  THEN 
 	M_PickPart := 1; // busy
	iGetPartSeq := 10;
	iConvReleasePartStatus := fbConveyorToPickFrom.M_ReleasePart(bReleasePartReq:=FALSE,bPartHandedOff:=FALSE); // Ask conveyor to release the part
END_IF

IF NOT bGetPart THEN 
	M_PickPart := 0 ; //idle, ready for next command
END_IF
CASE iGetPartSeq OF 
	0: (*Idle*)
		;
		
	10: (*Get part From Conveyor*)
		iConvReleasePartStatus := fbConveyorToPickFrom.M_ReleasePart(bReleasePartReq:=TRUE , bPartHandedOff:=FALSE, stPartToRelease=>stPart ); // Ask conveyor to release the part
		//if the part is non zero its ready take it 
		IF stPart.iIDNumber <>0 THEN 
			iGetPartSeq := 20;
			stPart.iCurrentDeviceID := P_DeviceID;
			bHavePart:=TRUE;
		END_IF
		IF iConvReleasePartStatus > 3 THEN // Function errored out
			fbConveyorToPickFrom.M_ReleasePart(bReleasePartReq:=FALSE, bPartHandedOff := FALSE); // Ask conveyor to release the part
			iGetPartSeq := 99;			
		END_IF
		
	20 : //Confirm receipt of part
		iConvReleasePartStatus := fbConveyorToPickFrom.M_ReleasePart(bReleasePartReq:=TRUE , bPartHandedOff:=TRUE); // Ask conveyor to release the part		
		IF iConvReleasePartStatus = 3 THEN 
			iGetPartSeq := 30;
		ELSIF iConvReleasePartStatus > 3 THEN
			iConvReleasePartStatus := fbConveyorToPickFrom.M_ReleasePart(bReleasePartReq:=FALSE , bPartHandedOff:=FALSE); // Ask conveyor to release the part		
			iGetPartSeq := 99;
		END_IF
	
	30: //Reset Request for part 	
		iConvReleasePartStatus := fbConveyorToPickFrom.M_ReleasePart(bReleasePartReq:=FALSE, bPartHandedOff := FALSE); // Ask conveyor to release the part
		IF iConvReleasePartStatus = 0 THEN 
			iGetPartSeq:= 0;
			M_PickPart := 3;
		END_IF
	99: //Error condition  
		eCurrentState := E_Error;
END_CASE
END_METHOD

METHOD PUBLIC M_PlacePart : UDINT
VAR_INPUT
	bPlacePart : BOOL;
END_VAR
VAR
END_VAR
fbTrigPlacePartSeq(CLK := bHavePart AND bPlacePart); 
IF fbTrigPlacePartSeq.Q THEN 
	M_PlacePart := 1;
	iPlacePartSeq:= 10;
END_IF
IF NOT bPlacePart THEN 
	 M_PlacePart := 0;
END_IF

CASE iPlacePartSeq OF
	0: (*Idle*)
	
	10: (*Find last part on Conveyor*)
		iConveyorAcceptStatus := fbConveyorToPlaceTo.M_AcceptPart(bPartPresentAtEntrance:=TRUE , stPartAtEntrance:=stPart );
		IF iConveyorAcceptStatus = 3 THEN 
			iPlacePartSeq := 20;
			iConveyorAcceptStatus := fbConveyorToPlaceTo.M_AcceptPart(bPartPresentAtEntrance:=FALSE , stPartAtEntrance:=stPart );
		END_IF
		IF iConveyorAcceptStatus > 3 THEN 
			iPlacePartSeq := 99;
			iConveyorAcceptStatus := fbConveyorToPlaceTo.M_AcceptPart(bPartPresentAtEntrance:=FALSE , stPartAtEntrance:=stPart );
		END_IF
	20:  //Hand the part to the requesting device
		stPart := stEmptyPart ; 
		bHavePart := FALSE;
		M_PlacePart := 0;
 
	99: //Error condition
		eCurrentState := E_Error;	
		
END_CASE
END_METHOD

END_FUNCTION_BLOCK

// ---- POUs/Sample OOP Conveyor/Device And Station Blocks/FB_Conveyor.TcPOU
FUNCTION_BLOCK FB_Conveyor EXTENDS FB_Device
VAR_INPUT
	bJogConveyorFwd : BOOL;
	bJogConveyorBwd : BOOL;
	fJogSpeed 		: LREAL;
	bRunConveyor	: BOOL;
	fCmdSpeed		: LREAL;
END_VAR
VAR_OUTPUT
	bReadyToAcceptPart 	: BOOL;
	bNotReadyToAcceptPart: BOOL;
	bPartInPickLocation : BOOL;
END_VAR
VAR_IN_OUT
	fbAxis				: I_Axis; //Pass the reference to ANY block that uses FB_Axis as a base class
END_VAR
VAR
	fbDisableConvSeq	: R_TRIG;
	fbDisableConvTrig	: R_TRIG;
	iDisableSeq			: INT;
	iAxisEnableState	: UDINT;
	iAxisResetState		: UDINT;
	fLastConveyorSpeed	: LREAL;
	iJogStatus			: UDINT;
	iAxisStopState		: UDINT;
	iAxisSpeedState		: UDINT;
	iDisableAxis		: UDINT;
	arrProductsOnConveyor: ARRAY [0..50] OF ST_PartData;
	fMinimumSpacing		: LREAL;
	fbTrigReleasePartSeq: R_TRIG;
	I					: INT;
	iReleasePartSeq		: INT;
	fPickLocation		: LREAL; 
	iLastPart			: INT;
	stEmptyPart			: ST_PartData;
	fCurrentSpeed 		: LREAL;
	fbNewSpeedTrig		: R_TRIG;
	fbNewCmdTrig		: R_TRIG;
	bIssueNewCommand	: BOOL;
END_VAR

(*States are selected according to method request*)
//Conveyor belt control
CASE eCurrentState OF
	E_Disabled: (*Disabled*)
		; 
	E_Error: (*Conveyor is in an Error State*)
		;
		
	E_Manual: (*Allow Manual commands to be called*)
		iJogStatus := fbAxis.M_Jog(bJogFwd:= bJogConveyorFwd, bJogBwd:= bJogConveyorBwd, fJogSpeed:=fJogSpeed );
		IF iJogStatus > 3 THEN 
			eCurrentState:= E_Error;
			iJogStatus:= fbAxis.M_Jog(bJogFwd:= FALSE, bJogBwd:= FALSE, fJogSpeed:=fJogSpeed );
		END_IF
		
	E_Auto:  (*Allow only automatic commands to be called*)
		iJogStatus:= fbAxis.M_Jog(bJogFwd:= FALSE, bJogBwd:= FALSE, fJogSpeed:=fJogSpeed );
		fbNewSpeedTrig(CLK:= (fCmdSpeed <> fLastConveyorSpeed) AND bRunConveyor);
		fbNewCmdTrig(CLK:= bRunConveyor);
		IF fbNewSpeedTrig.Q OR fbNewCmdTrig.Q THEN 
			bIssueNewCommand := TRUE;
		END_IF
		IF bIssueNewCommand AND iAxisSpeedState < 3 THEN 
			iAxisSpeedState := fbAxis.M_Speed(bMoveVelocity:=TRUE , fSpeed:=fCmdSpeed );
			fLastConveyorSpeed := fCmdSpeed;
		ELSIF iAxisSpeedState = 3 THEN 
			iAxisSpeedState :=fbAxis.M_Speed(bMoveVelocity:=FALSE , fSpeed:=fCmdSpeed );
			bIssueNewCommand := FALSE;
		ELSIF iAxisSpeedState > 3 THEN
			eCurrentState:=E_Error;
			iAxisSpeedState := fbAxis.M_Speed(bMoveVelocity:=FALSE , fSpeed:=fCmdSpeed );
			bIssueNewCommand := FALSE;
		END_IF			
		IF NOT bRunConveyor THEN 
			bIssueNewCommand := FALSE;
			iAxisSpeedState := fbAxis.M_Speed(bMoveVelocity:=FALSE , fSpeed:=fCmdSpeed );
		END_IF
END_CASE

//If there are any parts on the conveyor update their locations
bPartInPickLocation :=FALSE;
FOR I := 1 TO 50 DO
	IF arrProductsOnConveyor[I].fStartingConveyorPosition <> 0 THEN 
		arrProductsOnConveyor[I].fPosition := fbAxis.P_CurrentPosition - arrProductsOnConveyor[I].fStartingConveyorPosition;
		bPartInPickLocation := bPartInPickLocation OR (arrProductsOnConveyor[I].fPosition > fPickLocation );  
	END_IF
END_FOR

fCurrentSpeed := fbAxis.P_CurrentSpeed;

METHOD PUBLIC M_AcceptPart : UDINT
VAR_INPUT
	bPartPresentAtEntrance : BOOL;
	stPartAtEntrance : ST_PartData; 
END_VAR

VAR
	I: INT;
	fNextPartPosition: LREAL;
END_VAR
//If a part is present at the entrance determine if it can be accepted and if so accept 
IF bPartPresentAtEntrance THEN
	M_AcceptPart := 1; // Process is waiting 
	//Part can be accepted if it is far enough from the last part
	IF  (arrProductsOnConveyor[1].iIDNumber = 0)
	 OR (arrProductsOnConveyor[1].fPosition >  (stPartAtEntrance.fLength + fMinimumSpacing))  THEN
		//Shift all parts down one 
		 FOR I	:= 49 TO 2 BY -1 DO
			 arrProductsOnConveyor[I] := arrProductsOnConveyor[I-1];
		 END_FOR
		// after shifting add new part
		arrProductsOnConveyor[1] := stPartAtEntrance; 
		arrProductsOnConveyor[1].fStartingConveyorPosition:= fbAxis.P_CurrentPosition;
		arrProductsOnConveyor[1].iCurrentDeviceID := P_DeviceID;
		M_AcceptPart := 3; //Part has been accepted
	END_IF
END_IF
IF NOT bPartPresentAtEntrance THEN 
	M_AcceptPart := 0; //Idle
END_IF
END_METHOD

METHOD M_Auto : UDINT
VAR_INPUT
	bRequestAutoMode	: BOOL;
END_VAR
// Method confirms to the user it has complteted or that it is busy
// 0: idle
// 1: busy
// 3: complete
// > 3 Error condition
fbTrigAutoMode(CLK:= bRequestAutoMode);
IF fbTrigAutoMode.Q THEN
	iSwitchAutoSeq := 10;
	M_Auto:=1;
END_IF
IF NOT bRequestAutoMode THEN
	M_Auto:= 0;
END_IF

CASE iSwitchAutoSeq OF
	0: (*Idle*)
		;
	10: (*Verify all components can switch to Auto 
		Request all components to allow Auto*)
		eCurrentState:= E_SwitchingToAuto;
		iAxisEnableState := fbAxis.M_Enable(bEnable:=TRUE );
		iSwitchAutoSeq := 20;

	20:  (*Wait for all components to go to Auto*)
		iAxisEnableState := fbAxis.M_Enable(bEnable:=TRUE );
		IF iAxisEnableState =3 THEN (*If 3 then enable completed successfully*)
			iSwitchAutoSeq := 30;		
		ELSIF iAxisEnableState > 3 THEN (*If >3 error has been returned*)
			M_Auto := iAxisEnableState;
			iAxisEnableState := fbAxis.M_Enable(bEnable:=FALSE);
			iSwitchAutoSeq := 0;
		END_IF			 
	
	30: (*once all devices are in Auto confirm Auto mode*)
		eCurrentState := E_Auto;
		iSwitchAutoSeq := 0;
		M_Auto	:=3;	
		iAxisEnableState := fbAxis.M_Enable(bEnable:=FALSE);

END_CASE
END_METHOD

METHOD PUBLIC M_Disable : UDINT
VAR_INPUT
	bDisable: BOOL;
END_VAR
fbDisableConvTrig(CLK:=bDisable);
IF fbDisableConvTrig.Q THEN
	iDisableSeq := 10;
END_IF
IF NOT bDisable THEN
	M_Disable:= 0;
END_IF

CASE iDisableSeq OF
	0: (*Idle*)
		;
	10: 
		iDisableAxis := fbAxis.M_Disable(bDisable:=TRUE );
		IF iDisableAxis = 3 THEN
			iDisableSeq:= 20;
		END_IF
		
	20:
		iDisableAxis := fbAxis.M_Disable(bDisable:=FALSE );
		IF iDisableAxis = 0 THEN
			iDisableSeq:= 0;
		END_IF
END_CASE

IF iDisableAxis > 3 THEN 
	M_Disable := iDisableAxis;
	iDisableAxis := fbAxis.M_Disable(bDisable:=FALSE );
	iDisableSeq := 0;
END_IF
END_METHOD

METHOD M_Manual : UDINT
VAR_INPUT
	bRequestManualMode	: BOOL;
END_VAR
//The result of the method is an unsigned double integer
// 0 = idle 
// 1 = busy
// 3 = complete
// Any other number = Error
fbTrigManualMode(CLK:= bRequestManualMode);
IF fbTrigManualMode.Q THEN
	iSwitchManualSeq := 10;
	M_Manual:=1;
	(*Reset any methods or function blocks*)
	fbAxis.M_Reset(bReset:= TRUE);
	fbAxis.M_Enable(bEnable:=FALSE);
	fbAxis.M_Stop(bStop:= FALSE);
END_IF
IF NOT bRequestManualMode THEN
	M_Manual:= 0;
END_IF

CASE iSwitchManualSeq OF
	0: (*Idle*)
		;
	10: (*Check all components can switch to Manual*)
		eCurrentState:= E_SwitchingToManual;
		IF fbAxis.P_Error THEN (*If axis are errored, reset them*)
			iSwitchManualSeq := 20;
			iAxisResetState := fbAxis.M_Reset(bReset:= TRUE);
		ELSE 
			iSwitchManualSeq := 30;
		END_IF
		
			
	20: (*wait for reset to complete*)
		iAxisResetState := fbAxis.M_Reset(bReset:= TRUE);
		IF iAxisResetState = 3 THEN 
			iSwitchManualSeq := 30;
			iAxisResetState := fbAxis.M_Reset(bReset:= FALSE);
		ELSIF iAxisResetState > 3 THEN 
			M_Manual := iAxisResetState;
			iAxisResetState := fbAxis.M_Reset(bReset:= FALSE);
			iSwitchManualSeq := 0;		
		END_IF
	
	30:  (*ensure axis are enabled*)
		IF fbAxis.P_Ready THEN 
			iSwitchManualSeq := 50; 
		ELSE
			iAxisEnableState := fbAxis.M_Enable(bEnable:=TRUE );
			iSwitchManualSeq := 40;
		END_IF
	
	40: (*Wait for enables *)
		iAxisEnableState := fbAxis.M_Enable(bEnable:=TRUE );
		IF iAxisEnableState =3 THEN (*If 3 then enable completed successfully*)
			iSwitchManualSeq := 50;	
			iAxisEnableState := fbAxis.M_Enable(bEnable:=FALSE);
		ELSIF iAxisEnableState > 3 THEN (*If >3 error has been returned*)
			M_Manual := iAxisEnableState;
			iAxisEnableState := fbAxis.M_Enable(bEnable:=FALSE);
			iSwitchManualSeq := 0;
		END_IF			

	50: (*Ensure axis are stopped*) 
		IF ABS(fbAxis.P_CurrentSpeed) > 0.1 THEN 
			iAxisStopState := fbAxis.M_Stop(bStop:= TRUE) ;
			iSwitchManualSeq := 60; 
		ELSE 
			iSwitchManualSeq := 70; 	
		END_IF
		
	60: (*wait for axis to stop*)
		iAxisStopState := fbAxis.M_Stop(bStop:= TRUE) ;
		IF iAxisStopState = 3 THEN 
			iSwitchManualSeq := 70;
			iAxisStopState := fbAxis.M_Stop(bStop:= FALSE);	
		ELSIF iAxisStopState >3 THEN
			M_Manual:= iAxisStopState;
			iAxisStopState := fbAxis.M_Stop(bStop:= FALSE);
			iSwitchManualSeq:= 0;
		END_IF	
		
	70: (*once all devices are in Manual confirm Manual mode*)
		eCurrentState := E_Manual;
		iSwitchManualSeq := 0;
		M_Manual:=3;


END_CASE
END_METHOD

METHOD PUBLIC M_ReleasePart : UDINT
VAR_INPUT
	bReleasePartReq : BOOL; //Requested to release a part
	bPartHandedOff : BOOL; //Confirmation part has been taken
END_VAR
VAR_OUTPUT	
	stPartToRelease : ST_PartData;  //Part being released
END_VAR
VAR
	I: INT;  // I is a local variable 

END_VAR
fbTrigReleasePartSeq(CLK:=bReleasePartReq AND bPartInPickLocation); 
IF fbTrigReleasePartSeq.Q THEN 
	M_ReleasePart := 1;
	iReleasePartSeq:= 10; 
END_IF
IF NOT bReleasePartReq THEN 
	 M_ReleasePart := 0;
END_IF

CASE iReleasePartSeq OF
	0: (*Idle*)
	
	10: (*Find last part on Conveyor*)
		iLastPart :=0; 
		FOR I := 1 TO 50 DO 
			//Go through the list of parts find the last one that is present
			IF arrProductsOnConveyor[I].fLength > 0 THEN 
				iLastPart := I;  
			END_IF
		END_FOR
		IF iLastPart > 0 THEN
			iReleasePartSeq := 20;
		ELSE //no parts on conveyor
			iReleasePartSeq := 99; 
			eCurrentState := E_Error;
		END_IF	
	
	20:  //Hand the part to the requesting device
		stPartToRelease := arrProductsOnConveyor[iLastPart];
		IF bPartHandedOff THEN 
			iReleasePartSeq := 30;
		END_IF
		
	30: 
		arrProductsOnConveyor[iLastPart] := stEmptyPart;
		M_ReleasePart := 3;	
		iReleasePartSeq := 0; 
		
	99: 
		eCurrentState := E_Error;
END_CASE
END_METHOD

METHOD M_Reset : UDINT
VAR_INPUT
	bRequestReset	: BOOL;
END_VAR

VAR
	fbTrigReset: R_TRIG;
	iResetSeq: INT;
END_VAR
fbTrigReset(CLK:= bRequestReset);
IF fbTrigReset.Q THEN
	iResetSeq := 10;
	M_Reset:=1;
END_IF

CASE iResetSeq OF
	0: (*Idle*)
		;
	10: (*Request all sub devices to reset*)
		iResetSeq := 20;
		eCurrentState:= E_Resetting;
		iAxisResetState := fbAxis.M_Reset(bReset:=TRUE);
		
	20: //Call the methods to update the variables
		iAxisResetState := fbAxis.M_Reset(bReset:=TRUE);
		(*If axis reset state = 3 the reset is complete*)
		IF iAxisResetState = 3 THEN
			iResetSeq:= 30;
		ELSE
			M_Reset := iAxisResetState;
			iAxisResetState := fbAxis.M_Reset(bReset:=FALSE);
			iResetSeq:=0;			
		END_IF
	
	30: (*once all devices are in Manual confirm Manual mode*)
		eCurrentState := E_Reset;
		iResetSeq := 0;
		M_Reset:=3;
END_CASE
END_METHOD

PROPERTY PUBLIC P_MinimumSpacing : LREAL
GET
P_MinimumSpacing := fMinimumSpacing;
END_GET
SET
fMinimumSpacing := P_MinimumSpacing;
END_SET
END_PROPERTY

PROPERTY PUBLIC P_PickLocation : LREAL
GET
P_PickLocation :=  fPickLocation;
END_GET
SET
IF P_PickLocation > 0 THEN 
	fPickLocation := P_PickLocation;
END_IF
END_SET
END_PROPERTY

PROPERTY PUBLIC P_StartLocation : LREAL
GET
END_GET
SET
END_SET
END_PROPERTY

END_FUNCTION_BLOCK

// ---- POUs/GeneralPlcBlocks/FB_GenerateData.TcPOU
FUNCTION_BLOCK FB_GenerateData
VAR
	bTest			: BOOL;	
{attribute 'TcScope' := '< LineWidth:3, Color:green>'}
{attribute 'BaseUnit' := '<Frequency, 1, 0, 0>'}
	iTest			: INT;
	forward			: BOOL:=TRUE;
	bCheck			: BOOL := TRUE;
	iRadio			: INT;
END_VAR
VAR_OUTPUT
	strText			: STRING;	
	t				: UINT;
	Treppe			: INT;
	Rampe_Fast		: REAL;
	Rampe_Slow		: LREAL;
	i				: UINT;
	
	Peak			: LREAL;
	GrowSlow		: REAL;
	iCounter 		: DINT;
	Cosinus_Half	: LREAL;
	Sinus_Fast		: LREAL;
	Sinus_Slow1		: LREAL;
	Sinus_Slow2		: LREAL;
	Sinus_VerySlow	: LREAL;
	Sinus_SqFast	: LREAL;
	Sinus_SqSlow	: REAL;
	Sinus_Cos_Half	: LREAL;
	SinglePeak		: LREAL;
	phi				: REAL;
	Ts				: UINT;
	Rechteck1_1		: BOOL;
	Rechteck2_1		: BOOL;
	Rechteck3_1		: BOOL;

	Puls1			: REAL;
	Puls2			: REAL;

	dreieck			: REAL:=0;
	j				: UINT:=1;
	k				: UINT:=0;
	iValue			: INT;
	iValueBegin		: INT;
	iValueEnd		: INT;
	iValueArr		: ARRAY [0..100] OF DINT;
	iValueArr2		: ARRAY [0..2,0..10] OF DINT;
	
	bRed			: BOOL;
	bGreen			: BOOL;
	bYellow			: BOOL;
	bBlue			: BOOL;
	bGray			: BOOL;
	bBlue2			: BOOL;
	bGray2			: BOOL;
END_VAR


//Toggle based on number of cycle counts
t := t + 1;
iTest := iTest + 1;
IF iTest = 2500 THEN
	bTest := TRUE;
ELSIF iTest = 5000 THEN
	bTest := FALSE;
	iTest := 0;
END_IF

i:=i+1;
Ts:=128*10;
SinglePeak:=0;
IF (t>=2*Ts) THEN
	j:=j+1;
	t:=t-2*Ts;
END_IF

phi:=t/Ts;
Cosinus_Half:=COS(PI*t/(2*Ts));
Sinus_VerySlow:=COS(1*PI*(t)/Ts);
Sinus_Slow1:=COS(4*PI* (t+Ts/4+phi)/Ts);
Sinus_Slow2:= 0.000001*COS(4*PI* (t+Ts/3+phi)/Ts);
Sinus_Fast:=COS(12*PI*t/Ts);
Sinus_SqFast:=Sinus_Fast* Sinus_Slow1;
Sinus_SqSlow:=LREAL_TO_REAL(Sinus_VerySlow*Sinus_Slow1);

Sinus_Cos_Half:=(Cosinus_Half+Sinus_Slow2)*Sinus_SqSlow;
Rampe_Fast:=Rampe_Fast+0.1;

IF (Rampe_Fast>10.0) THEN
	Rampe_Fast:=-10.0;
END_IF

IF (t=0) THEN
	Rechteck1_1:=TRUE;
	Rechteck2_1:=TRUE;
	Rechteck3_1:=TRUE;
ELSIF (t=Ts/2) THEN
	Rechteck1_1:=FALSE;
ELSIF (t=Ts) THEN
	Rechteck1_1:=TRUE;
	Rechteck2_1:=FALSE;
ELSIF (t=3*Ts/2) THEN
	Rechteck1_1:=FALSE;
	Rechteck3_1:=FALSE;
END_IF

IF(i>250) THEN
	i:=0;
	Treppe:=Treppe+1;
END_IF

IF (Treppe>25) THEN
	Treppe:=0;
	SinglePeak:=1;
END_IF

IF (j>=1) THEN
	j:=0;
	forward:= NOT forward;
END_IF

IF (forward) THEN
	dreieck:=dreieck+0.002;
ELSE
	dreieck:=dreieck-0.002;
END_IF

Puls1:=LREAL_TO_REAL(Sinus_Fast*Sinus_VerySlow);
Puls2:=LREAL_TO_REAL(Sinus_SqSlow*Sinus_Fast);

Peak:=EXP(t*0.005)/10000;

k:=k+1;

IF (k>7) THEN
	k:=0;
	GrowSlow:=GrowSlow+(Sinus_SqSlow *(Puls1*Puls2*(Treppe+1)*0.01));
END_IF

iValueArr[iValue] := (iValueArr[iValue] + 1) MOD 101; 
iValueArr2[iValue MOD 3, iValue MOD 11] := (iValueArr[iValue] + 1) MOD 101; 

IF bCheck THEN
	CASE iRadio OF
		0: iValue := ABS(LREAL_TO_INT(100*Sinus_Slow1) MOD 101);
			iValueBegin := ABS(LREAL_TO_INT(100*Sinus_Fast) MOD 101); 
			iValueEnd := ABS(LREAL_TO_INT(100*Sinus_Slow1) MOD 101); 
		1: iValue := ABS(LREAL_TO_INT(100*Sinus_VerySlow) MOD 101);
			iValueBegin := ABS(LREAL_TO_INT(100*Sinus_Slow1) MOD 101); 
			iValueEnd := ABS(LREAL_TO_INT(100*Sinus_Fast) MOD 101); 
		2: iValue := ABS((Treppe * 10) MOD 101);
			iValueBegin := ABS(LREAL_TO_INT(100*Sinus_Fast) MOD 101); 
			iValueEnd := ABS(LREAL_TO_INT(100*Sinus_Fast + 50) MOD 101); 
	END_CASE

	bBlue			:= iValue > 20;
	bGray			:= iValue > 30;
	bYellow			:= iValue > 40;
	bGreen			:= iValue > 50;
	bBlue2			:= iValue > 60;
	bGray2			:= iValue > 70;
	bRed			:= iValue > 80;
	
END_IF

strText := CONCAT('Value: ', INT_TO_STRING(iValue));

END_FUNCTION_BLOCK

// ---- POUs/Sample UML SC/FB_UML_SC_Composite.TcPOU
FUNCTION_BLOCK FB_UML_SC_Composite
VAR	
	bInitFinished			: BOOL;
	bUseXmlFormat			: BOOL;
	bAllInfoCopiedToFile	: BOOL;
	bSendToMasterFinished	: BOOL;
	bSendToClientFinished	: BOOL;
END_VAR

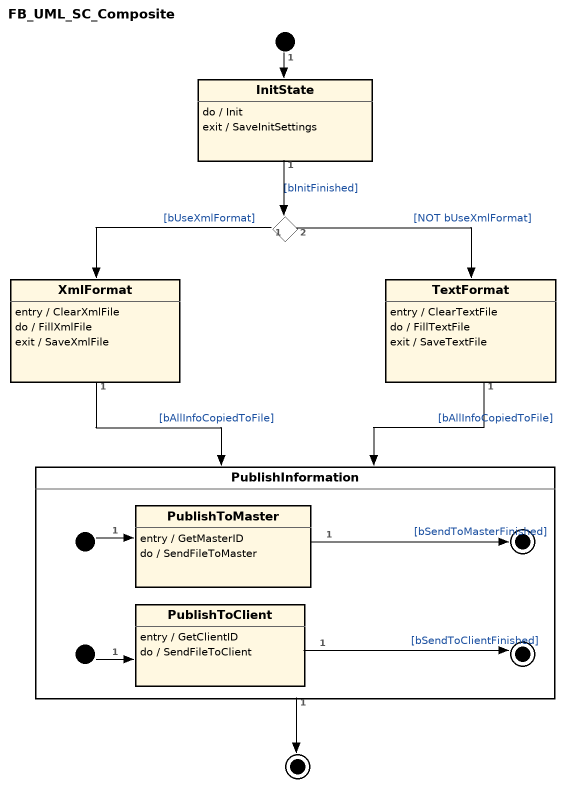
STATECHART FB_UML_SC_Composite  // abortable
    START StartState1
    STATE InitState
        do / Init
        exit / SaveInitSettings
    CHOICE ChoiceElement1
    STATE XmlFormat
        entry / ClearXmlFile
        do / FillXmlFile
        exit / SaveXmlFile
    STATE TextFormat
        entry / ClearTextFile
        do / FillTextFile
        exit / SaveTextFile
    COMPOSITE STATE PublishInformation
        REGION Region1 // priority 1
        START StartState3
        STATE PublishToClient
            entry / GetClientID
            do / SendFileToClient
        END EndState3
        StartState3 -> PublishToClient  // priority 1, on completion
        PublishToClient -> EndState3 [bSendToClientFinished] // priority 1
        REGION Region0 // priority 2
        START StartState2
        STATE PublishToMaster
            entry / GetMasterID
            do / SendFileToMaster
        END EndState2
        StartState2 -> PublishToMaster  // priority 1, on completion
        PublishToMaster -> EndState2 [bSendToMasterFinished] // priority 1
    END_STATE
    END EndState1
    StartState1 -> InitState  // priority 1, on completion
    InitState -> ChoiceElement1 [bInitFinished] // priority 1
    ChoiceElement1 -> XmlFormat [bUseXmlFormat] // priority 1
    ChoiceElement1 -> TextFormat [NOT bUseXmlFormat] // priority 2
    XmlFormat -> PublishInformation [bAllInfoCopiedToFile] // priority 1
    TextFormat -> PublishInformation [bAllInfoCopiedToFile] // priority 1
    PublishInformation -> EndState1  // priority 1, on completion
END_STATECHART

ACTION ClearTextFile:
nCounterClearText := nCounterClearText + 1;
END_ACTION

ACTION ClearXmlFile:
nCounterClearXml := nCounterClearXml + 1;
END_ACTION

ACTION FillTextFile:
nCounterFillText := nCounterFillText + 1;
END_ACTION

ACTION FillXmlFile:
nCounterFillXml := nCounterFillXml + 1;
END_ACTION

ACTION GetClientID:
nCounterGetClientID := nCounterGetClientID + 1;

IF nCounterGetClientID = 1 AND nCounterGetMasterID = 0 THEN
	bClientFirst := TRUE;
END_IF
END_ACTION

ACTION GetMasterID:
nCounterGetMasterID := nCounterGetMasterID + 1;

IF nCounterGetClientID = 0 AND nCounterGetMasterID = 1 THEN
	bMasterFirst := TRUE;
END_IF
END_ACTION

ACTION Init:
nCounterInit := nCounterInit + 1;
END_ACTION

ACTION SaveInitSettings:
nCounterSaveInitSettings := nCounterSaveInitSettings + 1;

bInitFinished 			:= FALSE;
bAllInfoCopiedToFile 	:= FALSE;
bSendToClientFinished 	:= FALSE;
bSendToMasterFinished	:= FALSE;
END_ACTION

ACTION SaveTextFile:
nCounterSaveText := nCounterSaveText + 1;
END_ACTION

ACTION SaveXmlFile:
nCounterSaveXml := nCounterSaveXml + 1;
END_ACTION

ACTION SendFileToClient:
nCounterSendToClient := nCounterSendToClient + 1;
END_ACTION

ACTION SendFileToMaster:
nCounterSendToMaster := nCounterSendToMaster + 1;
END_ACTION

END_FUNCTION_BLOCK

// ---- POUs/Sample UML SC/FB_UML_SC_Lamp.TcPOU
FUNCTION_BLOCK FB_UML_SC_Lamp
VAR_INPUT
	bPower				: BOOL;
END_VAR
VAR_OUTPUT
	ObLamp		AT%Q*	: BOOL;
END_VAR
VAR
	nCounterOn			: INT;
	nCounterOff			: INT;
END_VAR

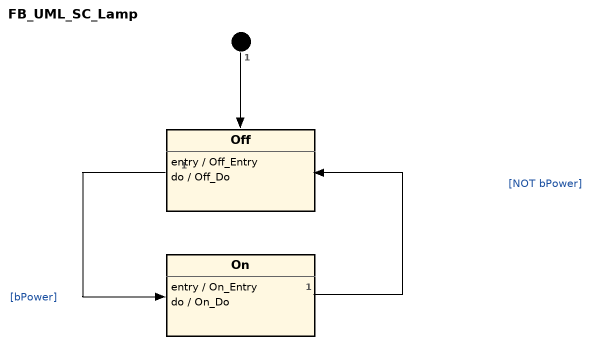
STATECHART FB_UML_SC_Lamp  // abortable
    START StartState1
    STATE Off
        entry / Off_Entry
        do / Off_Do
    STATE On
        entry / On_Entry
        do / On_Do
    StartState1 -> Off  // priority 1, on completion
    Off -> On [bPower] // priority 1, rising edge
    On -> Off [NOT bPower] // priority 1
END_STATECHART

ACTION Off_Do:
nCounterOff := nCounterOff + 1;
END_ACTION

ACTION Off_Entry:
ObLamp := FALSE;
END_ACTION

ACTION On_Do:
nCounterOn := nCounterOn + 1;
END_ACTION

ACTION On_Entry:
ObLamp := TRUE;
END_ACTION

END_FUNCTION_BLOCK

// ---- POUs/GeneralPlcBlocks/GeneralPlc.TcPOU
PROGRAM GeneralPlc
VAR
END_VAR
(* End *)

(* General *)

(* Analog input to output *)
	nAnalogOutP10 := nAnalogInR10;
	
(* Led on/off *)
	bLedH25 := bSwitchS25;

(* End *)

END_PROGRAM

// ---- POUs/GeneralPlcBlocks/Blinker.TcPOU
PROGRAM Blinker
VAR
	
	fbBlinker1								:FB_Blinker;
	tTurnOffDelayB1							:TIME := T#1S;
	fbBlinker2								:FB_Blinker;
	
END_VAR
(* End *)

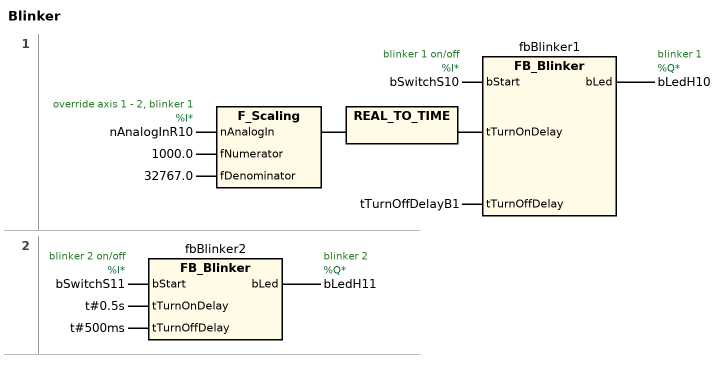
// NETWORK 1
//   bSwitchS10: blinker 1 on/off | AT %I*
//   nAnalogInR10: override axis 1 - 2, blinker 1 | AT %I*
//   bLedH10: blinker 1 | AT %Q*
fbBlinker1(
    bStart := bSwitchS10,
    tTurnOnDelay := REAL_TO_TIME(F_Scaling(nAnalogIn := nAnalogInR10, fNumerator := 1000.0, fDenominator := 32767.0)),
    tTurnOffDelay := tTurnOffDelayB1); // FB_Blinker
bLedH10 := fbBlinker1.bLed;

// NETWORK 2
//   bSwitchS11: blinker 2 on/off | AT %I*
//   bLedH11: blinker 2 | AT %Q*
fbBlinker2(bStart := bSwitchS11, tTurnOnDelay := t#0.5s, tTurnOffDelay := t#500ms); // FB_Blinker
bLedH11 := fbBlinker2.bLed;

END_PROGRAM

// ---- POUs/GeneralPlcBlocks/Components/FB_Blinker.TcPOU
FUNCTION_BLOCK FB_Blinker
VAR_INPUT

	bStart									:BOOL;
	tTurnOnDelay							:TIME;
	tTurnOffDelay							:TIME;

END_VAR
VAR_OUTPUT

	bLed									:BOOL;

END_VAR
VAR

	fbTimer1								:TON;
	fbTimer2								:TON;

END_VAR
(* End *)

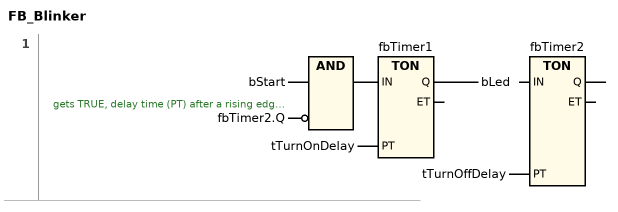
// NETWORK 1
//   fbTimer2.Q: gets TRUE, delay time (PT) after a rising edge at IN
fbTimer1(IN := bStart AND NOT fbTimer2.Q, PT := tTurnOnDelay); // TON
bLed := fbTimer1.Q;
fbTimer2(IN := fbTimer1.Q, PT := tTurnOffDelay); // TON

END_FUNCTION_BLOCK

// ---- POUs/GeneralPlcBlocks/Components/F_Scaling.TcPOU
FUNCTION F_Scaling : REAL
VAR_INPUT

	nAnalogIn								:INT;
	fNumerator								:REAL;
	fDenominator							:REAL;
	
END_VAR
VAR
END_VAR
(* End *)

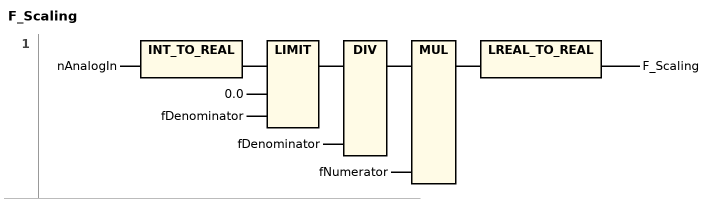
// NETWORK 1
F_Scaling := LREAL_TO_REAL((LIMIT(INT_TO_REAL(nAnalogIn), 0.0, fDenominator) / fDenominator) * fNumerator);

END_FUNCTION

// ---- POUs/GeneralPlcBlocks/ClockGenerator.TcPOU
PROGRAM ClockGenerator
VAR
	
	nCycleTime								:UDINT;		(* Cycle time from the PLC Task *)
	nTimeValue								:INT;		(* Time value clock generator*)
	
END_VAR
(* End *)

(* Clock generator *)

	(* PLC cycle time in ms  *)
	nCycleTime	:=	TwinCAT_SystemInfoVarList._TaskInfo[GETCURTASKINDEXEX()].cycleTime / 10000;

	(* Calculate with the cycle time the time value *)
	nTimeValue	:=	nTimeValue + UDINT_TO_INT(nCycleTime);

	(* Generate the clocks and the rising edges with the time value *)
	CASE nTimeValue OF

		500		:	bClock500ms			:=	TRUE;
					bRisingEdge500ms	:=	TRUE;

		1000	:	bClock500ms			:=	FALSE;
					bRisingEdge500ms	:=	TRUE;
					bClock1s			:=	TRUE;
					bRisingEdge1s		:=	TRUE;

		1500	:	bClock500ms			:=	TRUE;
					bRisingEdge500ms	:=	TRUE;

		2000	:	bClock500ms			:=	FALSE;
					bRisingEdge500ms	:=	TRUE;
					bClock1s			:=	FALSE;
					bRisingEdge1s		:=	TRUE;
					bClock2s			:=	TRUE;
					bRisingEdge2s		:=	TRUE;

		2500	:	bClock500ms			:=	TRUE;
					bRisingEdge500ms	:=	TRUE;

		3000	:	bClock500ms			:=	FALSE;
					bRisingEdge500ms	:=	TRUE;
					bClock1s			:=	TRUE;
					bRisingEdge1s		:=	TRUE;

		3500	:	bClock500ms			:=	TRUE;
					bRisingEdge500ms	:=	TRUE;

		4000	:	bClock500ms			:=	FALSE;
					bRisingEdge500ms	:=	TRUE;
			 		bClock1s			:=	FALSE;
					bRisingEdge1s		:=	TRUE;
					bClock2s			:=	FALSE;
					bRisingEdge2s		:=	TRUE;
					
	ELSE

		(* Reset the rising edge variables after one cycle *)
		bRisingEdge500ms	:=	FALSE;
		bRisingEdge1s		:=	FALSE;
		bRisingEdge2s		:=	FALSE;

	END_CASE;

	(* Sequence reset at 4000ms *)
	IF nTimeValue >= 4000
	THEN
		nTimeValue := 0;
	END_IF

(* End *)

END_PROGRAM

// ---- POUs/Motion/AxisGeneral.TcPOU
PROGRAM AxisGeneral
VAR
	
	bAxis3ReferenceCam						:BOOL;
	bAxis4ReferenceCam						:BOOL;

END_VAR
(* End *)

(* Axis general *)

(* EL7037 *)
	(* Reference cam Axis 1 *)
	bStepperReferenceCam;

(* EL7201 *)
	(* Reference cam Axis 2 *)
	bAxis2ReferenceCamEL7;

(* AX5203 *)
	(* Reference cam Axis 3 *)
	bLedH26 				:= nAX5203DigitalInputs.0;
	bAxis3ReferenceCam		:= nAX5203DigitalInputs.0;

	(* Reference cam Axis 4 *)
	nAX5203DigitalOutputs.7 := nAX5203DigitalInputs.1;
	bAxis4ReferenceCam		:= nAX5203DigitalInputs.1;
	
	(* Switch S26 *)
	nAX5203DigitalInputs.2;

